   LIN {X 0.148, Y -17.815, Z 116.450} C_DIS
   LIN {X 0.105, Y -17.697, Z 116.450} C_DIS
   LIN {X 0.144, Y -15.870, Z 116.450} C_DIS
   LIN {X 0.185, Y -15.606, Z 116.450} C_DIS
   LIN {X 0.334, Y -15.400, Z 116.450} C_DIS
   LIN {X 1.468, Y -13.305, Z 116.450} C_DIS
   LIN {X 2.152, Y -12.926, Z 116.450} C_DIS
   LIN {X 3.732, Y -11.958, Z 116.450} C_DIS
   LIN {X 5.275, Y -11.875, Z 116.450} C_DIS
   LIN {X 5.904, Y -11.838, Z 116.450} C_DIS
   LIN {X 6.625, Y -12.128, Z 116.450} C_DIS
   LIN {X 7.876, Y -12.635, Z 116.450} C_DIS
   LIN {X 8.873, Y -13.791, Z 116.450} C_DIS
   LIN {X 9.540, Y -14.557, Z 116.450} C_DIS
   LIN {X 9.767, Y -15.717, Z 116.450}
   LaserEnd_Ext()
   LIN {X -10.909, Y 41.483, Z 116.450}
   LaserStart_Ext()
   LIN {X -11.006, Y 41.733, Z 116.450} C_DIS
   LIN {X -11.451, Y 43.299, Z 116.450} C_DIS
   LIN {X -10.985, Y 45.327, Z 116.450} C_DIS
   LIN {X -10.916, Y 45.490, Z 116.450} C_DIS
   LIN {X -10.671, Y 45.761, Z 116.450} C_DIS
   LIN {X -9.977, Y 46.585, Z 116.450} C_DIS
   LIN {X -9.388, Y 46.930, Z 116.450} C_DIS
   LIN {X -8.600, Y 47.307, Z 116.450} C_DIS
   LIN {X -8.343, Y 47.326, Z 116.450} C_DIS
   LIN {X -6.766, Y 47.399, Z 116.450} C_DIS
   LIN {X -6.451, Y 47.269, Z 116.450} C_DIS
   LIN {X -5.150, Y 46.712, Z 116.450} C_DIS
   LIN {X -4.172, Y 45.690, Z 116.450} C_DIS
   LIN {X -4.100, Y 45.595, Z 116.450} C_DIS
   LIN {X -3.202, Y 44.213, Z 116.450} C_DIS
   LIN {X -2.206, Y 42.575, Z 116.450} C_DIS
   LIN {X -1.280, Y 41.069, Z 116.450} C_DIS
   LIN {X 0.088, Y 38.632, Z 116.450} C_DIS
   LIN {X 0.776, Y 37.421, Z 116.450} C_DIS
   LIN {X 1.017, Y 36.980, Z 116.450} C_DIS
   LIN {X 3.124, Y 32.754, Z 116.450} C_DIS
   LIN {X 4.597, Y 29.710, Z 116.450} C_DIS
   LIN {X 5.895, Y 26.489, Z 116.450} C_DIS
   LIN {X 7.344, Y 22.915, Z 116.450} C_DIS
   LIN {X 8.835, Y 18.359, Z 116.450} C_DIS
   LIN {X 10.168, Y 14.012, Z 116.450} C_DIS
   LIN {X 11.828, Y 6.827, Z 116.450} C_DIS
   LIN {X 12.484, Y 3.575, Z 116.450} C_DIS
   LIN {X 13.461, Y -3.473, Z 116.450} C_DIS
   LIN {X 13.499, Y -3.785, Z 116.450} C_DIS
   LIN {X 13.808, Y -7.587, Z 116.450} C_DIS
   LIN {X 13.839, Y -7.818, Z 116.450} C_DIS
   LIN {X 13.902, Y -8.784, Z 116.450} C_DIS
   LIN {X 13.967, Y -10.194, Z 116.450} C_DIS
   LIN {X 14.021, Y -11.696, Z 116.450} C_DIS
   LIN {X 14.069, Y -13.595, Z 116.450} C_DIS
   LIN {X 14.061, Y -15.779, Z 116.450} C_DIS
   LIN {X 14.062, Y -16.860, Z 116.450} C_DIS
   LIN {X 13.686, Y -18.412, Z 116.450} C_DIS
   LIN {X 13.131, Y -20.708, Z 116.450} C_DIS
   LIN {X 12.132, Y -22.067, Z 116.450} C_DIS
   LIN {X 11.479, Y -23.029, Z 116.450} C_DIS
   LIN {X 10.917, Y -23.560, Z 116.450} C_DIS
   LIN {X 9.337, Y -24.637, Z 116.450} C_DIS
   LIN {X 8.125, Y -25.174, Z 116.450} C_DIS
   LIN {X 5.580, Y -25.760, Z 116.450} C_DIS
   LIN {X 4.678, Y -25.759, Z 116.450} C_DIS
   LIN {X 2.942, Y -25.575, Z 116.450} C_DIS
   LIN {X 2.640, Y -25.450, Z 116.450} C_DIS
   LIN {X -0.209, Y -24.162, Z 116.450} C_DIS
   LIN {X -0.493, Y -23.865, Z 116.450} C_DIS
   LIN {X -2.856, Y -21.202, Z 116.450} C_DIS
   LIN {X -3.165, Y -20.226, Z 116.450} C_DIS
   LIN {X -3.943, Y -17.598, Z 116.450} C_DIS
   LIN {X -3.816, Y -16.292, Z 116.450} C_DIS
   LIN {X -3.648, Y -14.441, Z 116.450} C_DIS
   LIN {X -2.859, Y -11.235, Z 116.450} C_DIS
   LIN {X -2.701, Y -10.616, Z 116.450} C_DIS
   LIN {X -2.627, Y -10.239, Z 116.450} C_DIS
   LIN {X -2.158, Y -7.884, Z 116.450} C_DIS
   LIN {X -1.604, Y -4.053, Z 116.450} C_DIS
   LIN {X -1.466, Y -3.109, Z 116.450} C_DIS
   LIN {X -1.367, Y -1.347, Z 116.450} C_DIS
   LIN {X -1.059, Y 3.657, Z 116.450} C_DIS
   LIN {X -1.134, Y 7.378, Z 116.450} C_DIS
   LIN {X -1.528, Y 13.286, Z 116.450} C_DIS
   LIN {X -2.342, Y 18.188, Z 116.450} C_DIS
   LIN {X -3.212, Y 22.624, Z 116.450} C_DIS
   LIN {X -4.479, Y 26.756, Z 116.450} C_DIS
   LIN {X -5.529, Y 30.144, Z 116.450} C_DIS
   LIN {X -5.798, Y 30.771, Z 116.450} C_DIS
   LIN {X -6.098, Y 31.534, Z 116.450} C_DIS
   LIN {X -7.395, Y 34.580, Z 116.450} C_DIS
   LIN {X -8.008, Y 35.958, Z 116.450} C_DIS
   LIN {X -8.997, Y 37.945, Z 116.450} C_DIS
   LIN {X -9.450, Y 38.841, Z 116.450} C_DIS
   LIN {X -10.064, Y 39.969, Z 116.450} C_DIS
   LIN {X -10.750, Y 41.198, Z 116.450} C_DIS
   LIN {X -10.909, Y 41.483, Z 116.450}
   LaserEnd_Ext()
   LIN {X 12.602, Y -5.091, Z 116.450}
   LaserStart_Ext()
   LIN {X 12.602, Y -18.640, Z 116.450}
   LaserEnd_Ext()
   LIN {X 11.602, Y -21.099, Z 116.450}
   LaserStart_Ext()
   LIN {X 11.602, Y 2.657, Z 116.450}
   LaserEnd_Ext()
   LIN {X 10.602, Y 7.690, Z 116.450}
   LaserStart_Ext()
   LIN {X 10.602, Y -14.776, Z 116.450}
   LaserEnd_Ext()
   LIN {X 10.602, Y -18.691, Z 116.450}
   LaserStart_Ext()
   LIN {X 10.602, Y -22.482, Z 116.450}
   LaserEnd_Ext()
   LIN {X 9.602, Y -23.246, Z 116.450}
   LaserStart_Ext()
   LIN {X 9.602, Y -20.491, Z 116.450}
   LaserEnd_Ext()
   LIN {X 9.602, Y -13.105, Z 116.450}
   LaserStart_Ext()
   LIN {X 9.602, Y 12.019, Z 116.450}
   LaserEnd_Ext()
   LIN {X 8.602, Y 15.708, Z 116.450}
   LaserStart_Ext()
   LIN {X 8.602, Y -11.949, Z 116.450}
   LaserEnd_Ext()
   LIN {X 8.602, Y -21.573, Z 116.450}
   LaserStart_Ext()
   LIN {X 8.602, Y -23.869, Z 116.450}
   LaserEnd_Ext()
   LIN {X 7.602, Y -24.269, Z 116.450}
   LaserStart_Ext()
   LIN {X 7.602, Y -22.068, Z 116.450}
   LaserEnd_Ext()
   LIN {X 7.602, Y -11.445, Z 116.450}
   LaserStart_Ext()
   LIN {X 7.602, Y 18.912, Z 116.450}
   LaserEnd_Ext()
   LIN {X 6.602, Y 21.967, Z 116.450}
   LaserStart_Ext()
   LIN {X 6.602, Y -11.041, Z 116.450}
   LaserEnd_Ext()
   LIN {X 6.602, Y -22.559, Z 116.450}
   LaserStart_Ext()
   LIN {X 6.602, Y -24.499, Z 116.450}
   LaserEnd_Ext()
   LIN {X 5.602, Y -24.728, Z 116.450}
   LaserStart_Ext()
   LIN {X 5.602, Y -22.670, Z 116.450}
   LaserEnd_Ext()
   LIN {X 5.602, Y -10.854, Z 116.450}
   LaserStart_Ext()
   LIN {X 5.602, Y 24.551, Z 116.450}
   LaserEnd_Ext()
   LIN {X 4.602, Y 27.023, Z 116.450}
   LaserStart_Ext()
   LIN {X 4.602, Y -10.910, Z 116.450}
   LaserEnd_Ext()
   LIN {X 4.602, Y -22.710, Z 116.450}
   LaserStart_Ext()
   LIN {X 4.602, Y -24.745, Z 116.450}
   LaserEnd_Ext()
   LIN {X 3.602, Y -24.639, Z 116.450}
   LaserStart_Ext()
   LIN {X 3.602, Y -22.581, Z 116.450}
   LaserEnd_Ext()
   LIN {X 3.602, Y -10.967, Z 116.450}
   LaserStart_Ext()
   LIN {X 3.602, Y 29.471, Z 116.450}
   LaserEnd_Ext()
   LIN {X 2.602, Y 31.537, Z 116.450}
   LaserStart_Ext()
   LIN {X 2.602, Y -11.477, Z 116.450}
   LaserEnd_Ext()
   LIN {X 2.602, Y -22.181, Z 116.450}
   LaserStart_Ext()
   LIN {X 2.602, Y -24.335, Z 116.450}
   LaserEnd_Ext()
   LIN {X 1.602, Y -23.883, Z 116.450}
   LaserStart_Ext()
   LIN {X 1.602, Y -21.731, Z 116.450}
   LaserEnd_Ext()
   LIN {X 1.602, Y -12.088, Z 116.450}
   LaserStart_Ext()
   LIN {X 1.602, Y 33.566, Z 116.450}
   LaserEnd_Ext()
   LIN {X 0.602, Y 35.571, Z 116.450}
   LaserStart_Ext()
   LIN {X 0.602, Y -12.808, Z 116.450}
   LaserEnd_Ext()
   LIN {X 0.602, Y -20.717, Z 116.450}
   LaserStart_Ext()
   LIN {X 0.602, Y -23.432, Z 116.450}
   LaserEnd_Ext()
   LIN {X -0.398, Y -22.465, Z 116.450}
   LaserStart_Ext()
   LIN {X -0.398, Y -19.184, Z 116.450}
   LaserEnd_Ext()
   LIN {X -0.398, Y -14.651, Z 116.450}
   LaserStart_Ext()
   LIN {X -0.398, Y -1.923, Z 116.450}
   LaserEnd_Ext()
   LIN {X -0.398, Y 11.377, Z 116.450}
   LaserStart_Ext()
   LIN {X -0.398, Y 37.462, Z 116.450}
   LaserEnd_Ext()
   LIN {X -1.398, Y 39.236, Z 116.450}
   LaserStart_Ext()
   LIN {X -1.398, Y 18.572, Z 116.450}
   LaserEnd_Ext()
   LIN {X -1.398, Y -9.189, Z 116.450}
   LaserStart_Ext()
   LIN {X -1.398, Y -21.338, Z 116.450}
   LaserEnd_Ext()
   LIN {X -2.398, Y -19.295, Z 116.450}
   LaserStart_Ext()
   LIN {X -2.398, Y -13.547, Z 116.450}
   LaserEnd_Ext()
   LIN {X -2.398, Y 23.380, Z 116.450}
   LaserStart_Ext()
   LIN {X -2.398, Y 40.979, Z 116.450}
   LaserEnd_Ext()
   LIN {X -3.398, Y 42.611, Z 116.450}
   LaserStart_Ext()
   LIN {X -3.398, Y 26.642, Z 116.450}
   LaserEnd_Ext()
   LIN {X -4.398, Y 29.872, Z 116.450}
   LaserStart_Ext()
   LIN {X -4.398, Y 44.218, Z 116.450}
   LaserEnd_Ext()
   LIN {X -5.398, Y 45.524, Z 116.450}
   LaserStart_Ext()
   LIN {X -5.398, Y 32.443, Z 116.450}
   LaserEnd_Ext()
   LIN {X -6.398, Y 34.792, Z 116.450}
   LaserStart_Ext()
   LIN {X -6.398, Y 46.158, Z 116.450}
   LaserEnd_Ext()
   LIN {X -7.398, Y 46.368, Z 116.450}
   LaserStart_Ext()
   LIN {X -7.398, Y 36.977, Z 116.450}
   LaserEnd_Ext()
   LIN {X -8.398, Y 38.977, Z 116.450}
   LaserStart_Ext()
   LIN {X -8.398, Y 46.295, Z 116.450}
   LaserEnd_Ext()
   LIN {X -9.398, Y 45.720, Z 116.450}
   LaserStart_Ext()
   LIN {X -9.398, Y 40.828, Z 116.450}
   LaserEnd_Ext()
   LIN {X -10.398, Y 43.252, Z 116.450}
   LaserStart_Ext()
   LIN {X -10.398, Y 43.501, Z 116.450}
   LaserEnd_Ext()
   LIN {X 2.352, Y -12.792, Z 117.300}
   LaserStart_Ext()
   LIN {X 3.808, Y -11.899, Z 117.300} C_DIS
   LIN {X 4.082, Y -11.884, Z 117.300} C_DIS
   LIN {X 5.981, Y -11.774, Z 117.300} C_DIS
   LIN {X 7.781, Y -12.497, Z 117.300} C_DIS
   LIN {X 7.954, Y -12.566, Z 117.300} C_DIS
   LIN {X 8.122, Y -12.758, Z 117.300} C_DIS
   LIN {X 9.624, Y -14.482, Z 117.300} C_DIS
   LIN {X 10.019, Y -16.502, Z 117.300} C_DIS
   LIN {X 10.117, Y -17.066, Z 117.300} C_DIS
   LIN {X 10.008, Y -17.325, Z 117.300} C_DIS
   LIN {X 9.461, Y -19.163, Z 117.300} C_DIS
   LIN {X 9.174, Y -19.483, Z 117.300} C_DIS
   LIN {X 8.261, Y -20.603, Z 117.300} C_DIS
   LIN {X 7.039, Y -21.215, Z 117.300} C_DIS
   LIN {X 6.305, Y -21.578, Z 117.300} C_DIS
   LIN {X 5.059, Y -21.630, Z 117.300} C_DIS
   LIN {X 4.256, Y -21.666, Z 117.300} C_DIS
   LIN {X 3.735, Y -21.461, Z 117.300} C_DIS
   LIN {X 2.335, Y -20.902, Z 117.300} C_DIS
   LIN {X 1.034, Y -19.575, Z 117.300} C_DIS
   LIN {X 0.886, Y -19.430, Z 117.300} C_DIS
   LIN {X 0.843, Y -19.336, Z 117.300} C_DIS
   LIN {X 0.209, Y -17.706, Z 117.300} C_DIS
   LIN {X 0.242, Y -16.089, Z 117.300} C_DIS
   LIN {X 0.232, Y -15.677, Z 117.300} C_DIS
   LIN {X 1.388, Y -13.470, Z 117.300} C_DIS
   LIN {X 1.506, Y -13.295, Z 117.300} C_DIS
   LIN {X 2.352, Y -12.792, Z 117.300}
   LaserEnd_Ext()
   LIN {X -10.228, Y 46.455, Z 117.300}
   LaserStart_Ext()
   LIN {X -8.835, Y 47.270, Z 117.300} C_DIS
   LIN {X -8.739, Y 47.316, Z 117.300} C_DIS
   LIN {X -7.015, Y 47.441, Z 117.300} C_DIS
   LIN {X -6.906, Y 47.446, Z 117.300} C_DIS
   LIN {X -5.837, Y 47.004, Z 117.300} C_DIS
   LIN {X -5.218, Y 46.751, Z 117.300} C_DIS
   LIN {X -4.194, Y 45.692, Z 117.300} C_DIS
   LIN {X -3.623, Y 44.809, Z 117.300} C_DIS
   LIN {X -3.110, Y 44.019, Z 117.300} C_DIS
   LIN {X -1.466, Y 41.317, Z 117.300} C_DIS
   LIN {X -1.246, Y 40.962, Z 117.300} C_DIS
   LIN {X -1.128, Y 40.764, Z 117.300} C_DIS
   LIN {X 0.502, Y 37.895, Z 117.300} C_DIS
   LIN {X 1.213, Y 36.595, Z 117.300} C_DIS
   LIN {X 2.850, Y 33.312, Z 117.300} C_DIS
   LIN {X 4.633, Y 29.628, Z 117.300} C_DIS
   LIN {X 5.665, Y 27.069, Z 117.300} C_DIS
   LIN {X 7.447, Y 22.670, Z 117.300} C_DIS
   LIN {X 8.661, Y 18.962, Z 117.300} C_DIS
   LIN {X 10.345, Y 13.469, Z 117.300} C_DIS
   LIN {X 11.735, Y 7.454, Z 117.300} C_DIS
   LIN {X 12.611, Y 3.117, Z 117.300} C_DIS
   LIN {X 13.446, Y -2.907, Z 117.300} C_DIS
   LIN {X 13.600, Y -4.184, Z 117.300} C_DIS
   LIN {X 13.868, Y -7.474, Z 117.300} C_DIS
   LIN {X 13.906, Y -7.768, Z 117.300} C_DIS
   LIN {X 13.987, Y -8.999, Z 117.300} C_DIS
   LIN {X 14.014, Y -9.585, Z 117.300} C_DIS
   LIN {X 14.134, Y -12.868, Z 117.300} C_DIS
   LIN {X 14.150, Y -13.509, Z 117.300} C_DIS
   LIN {X 14.147, Y -14.246, Z 117.300} C_DIS
   LIN {X 14.152, Y -16.774, Z 117.300} C_DIS
   LIN {X 13.271, Y -20.403, Z 117.300} C_DIS
   LIN {X 13.205, Y -20.676, Z 117.300} C_DIS
   LIN {X 13.086, Y -20.838, Z 117.300} C_DIS
   LIN {X 11.830, Y -22.691, Z 117.300} C_DIS
   LIN {X 10.750, Y -23.712, Z 117.300} C_DIS
   LIN {X 9.871, Y -24.310, Z 117.300} C_DIS
   LIN {X 7.645, Y -25.298, Z 117.300} C_DIS
   LIN {X 6.126, Y -25.647, Z 117.300} C_DIS
   LIN {X 4.190, Y -25.646, Z 117.300} C_DIS
   LIN {X 3.126, Y -25.533, Z 117.300} C_DIS
   LIN {X 1.700, Y -24.941, Z 117.300} C_DIS
   LIN {X -0.040, Y -24.154, Z 117.300} C_DIS
   LIN {X -1.305, Y -22.829, Z 117.300} C_DIS
   LIN {X -2.695, Y -21.263, Z 117.300} C_DIS
   LIN {X -3.641, Y -18.277, Z 117.300} C_DIS
   LIN {X -3.853, Y -17.560, Z 117.300} C_DIS
   LIN {X -3.818, Y -17.203, Z 117.300} C_DIS
   LIN {X -3.565, Y -14.402, Z 117.300} C_DIS
   LIN {X -2.820, Y -11.378, Z 117.300} C_DIS
   LIN {X -2.522, Y -10.037, Z 117.300} C_DIS
   LIN {X -2.151, Y -8.171, Z 117.300} C_DIS
   LIN {X -1.440, Y -3.250, Z 117.300} C_DIS
   LIN {X -1.418, Y -3.006, Z 117.300} C_DIS
   LIN {X -1.034, Y 3.218, Z 117.300} C_DIS
   LIN {X -1.127, Y 7.848, Z 117.300} C_DIS
   LIN {X -1.461, Y 12.849, Z 117.300} C_DIS
   LIN {X -2.442, Y 18.758, Z 117.300} C_DIS
   LIN {X -3.160, Y 22.418, Z 117.300} C_DIS
   LIN {X -4.659, Y 27.305, Z 117.300} C_DIS
   LIN {X -5.505, Y 30.034, Z 117.300} C_DIS
   LIN {X -5.809, Y 30.745, Z 117.300} C_DIS
   LIN {X -5.975, Y 31.166, Z 117.300} C_DIS
   LIN {X -7.620, Y 35.030, Z 117.300} C_DIS
   LIN {X -7.914, Y 35.691, Z 117.300} C_DIS
   LIN {X -9.253, Y 38.384, Z 117.300} C_DIS
   LIN {X -9.442, Y 38.756, Z 117.300} C_DIS
   LIN {X -9.697, Y 39.225, Z 117.300} C_DIS
   LIN {X -10.133, Y 40.006, Z 117.300} C_DIS
   LIN {X -10.961, Y 41.508, Z 117.300} C_DIS
   LIN {X -11.151, Y 42.020, Z 117.300} C_DIS
   LIN {X -11.490, Y 43.166, Z 117.300} C_DIS
   LIN {X -11.440, Y 43.879, Z 117.300} C_DIS
   LIN {X -11.089, Y 45.273, Z 117.300} C_DIS
   LIN {X -10.777, Y 45.775, Z 117.300} C_DIS
   LIN {X -10.454, Y 46.186, Z 117.300} C_DIS
   LIN {X -10.228, Y 46.455, Z 117.300}
   LaserEnd_Ext()
   LIN {X -9.705, Y 45.522, Z 117.300}
   LaserStart_Ext()
   LIN {X -5.421, Y 45.522, Z 117.300}
   LaserEnd_Ext()
   LIN {X -4.628, Y 44.522, Z 117.300}
   LaserStart_Ext()
   LIN {X -10.247, Y 44.522, Z 117.300}
   LaserEnd_Ext()
   LIN {X -10.463, Y 43.522, Z 117.300}
   LaserStart_Ext()
   LIN {X -3.979, Y 43.522, Z 117.300}
   LaserEnd_Ext()
   LIN {X -3.369, Y 42.522, Z 117.300}
   LaserStart_Ext()
   LIN {X -10.257, Y 42.522, Z 117.300}
   LaserEnd_Ext()
   LIN {X -9.827, Y 41.522, Z 117.300}
   LaserStart_Ext()
   LIN {X -2.761, Y 41.522, Z 117.300}
   LaserEnd_Ext()
   LIN {X -2.150, Y 40.522, Z 117.300}
   LaserStart_Ext()
   LIN {X -9.275, Y 40.522, Z 117.300}
   LaserEnd_Ext()
   LIN {X -8.720, Y 39.522, Z 117.300}
   LaserStart_Ext()
   LIN {X -1.573, Y 39.522, Z 117.300}
   LaserEnd_Ext()
   LIN {X -1.004, Y 38.522, Z 117.300}
   LaserStart_Ext()
   LIN {X -8.205, Y 38.522, Z 117.300}
   LaserEnd_Ext()
   LIN {X -7.708, Y 37.522, Z 117.300}
   LaserStart_Ext()
   LIN {X -0.436, Y 37.522, Z 117.300}
   LaserEnd_Ext()
   LIN {X 0.114, Y 36.522, Z 117.300}
   LaserStart_Ext()
   LIN {X -7.210, Y 36.522, Z 117.300}
   LaserEnd_Ext()
   LIN {X -6.744, Y 35.522, Z 117.300}
   LaserStart_Ext()
   LIN {X 0.631, Y 35.522, Z 117.300}
   LaserEnd_Ext()
   LIN {X 1.130, Y 34.522, Z 117.300}
   LaserStart_Ext()
   LIN {X -6.317, Y 34.522, Z 117.300}
   LaserEnd_Ext()
   LIN {X -5.891, Y 33.522, Z 117.300}
   LaserStart_Ext()
   LIN {X 1.628, Y 33.522, Z 117.300}
   LaserEnd_Ext()
   LIN {X 2.122, Y 32.522, Z 117.300}
   LaserStart_Ext()
   LIN {X -5.465, Y 32.522, Z 117.300}
   LaserEnd_Ext()
   LIN {X -5.040, Y 31.522, Z 117.300}
   LaserStart_Ext()
   LIN {X 2.606, Y 31.522, Z 117.300}
   LaserEnd_Ext()
   LIN {X 3.090, Y 30.522, Z 117.300}
   LaserStart_Ext()
   LIN {X -4.626, Y 30.522, Z 117.300}
   LaserEnd_Ext()
   LIN {X -4.299, Y 29.522, Z 117.300}
   LaserStart_Ext()
   LIN {X 3.574, Y 29.522, Z 117.300}
   LaserEnd_Ext()
   LIN {X 4.001, Y 28.522, Z 117.300}
   LaserStart_Ext()
   LIN {X -3.989, Y 28.522, Z 117.300}
   LaserEnd_Ext()
   LIN {X -3.679, Y 27.522, Z 117.300}
   LaserStart_Ext()
   LIN {X 4.404, Y 27.522, Z 117.300}
   LaserEnd_Ext()
   LIN {X 4.808, Y 26.522, Z 117.300}
   LaserStart_Ext()
   LIN {X -3.373, Y 26.522, Z 117.300}
   LaserEnd_Ext()
   LIN {X -3.066, Y 25.522, Z 117.300}
   LaserStart_Ext()
   LIN {X 5.213, Y 25.522, Z 117.300}
   LaserEnd_Ext()
   LIN {X 5.618, Y 24.522, Z 117.300}
   LaserStart_Ext()
   LIN {X -2.760, Y 24.522, Z 117.300}
   LaserEnd_Ext()
   LIN {X -2.453, Y 23.522, Z 117.300}
   LaserStart_Ext()
   LIN {X 6.023, Y 23.522, Z 117.300}
   LaserEnd_Ext()
   LIN {X 6.429, Y 22.522, Z 117.300}
   LaserStart_Ext()
   LIN {X -2.162, Y 22.522, Z 117.300}
   LaserEnd_Ext()
   LIN {X -1.966, Y 21.522, Z 117.300}
   LaserStart_Ext()
   LIN {X 6.771, Y 21.522, Z 117.300}
   LaserEnd_Ext()
   LIN {X 7.098, Y 20.522, Z 117.300}
   LaserStart_Ext()
   LIN {X -1.769, Y 20.522, Z 117.300}
   LaserEnd_Ext()
   LIN {X -1.573, Y 19.522, Z 117.300}
   LaserStart_Ext()
   LIN {X 7.426, Y 19.522, Z 117.300}
   LaserEnd_Ext()
   LIN {X 7.750, Y 18.522, Z 117.300}
   LaserStart_Ext()
   LIN {X -1.389, Y 18.522, Z 117.300}
   LaserEnd_Ext()
   LIN {X -1.223, Y 17.522, Z 117.300}
   LaserStart_Ext()
   LIN {X 8.057, Y 17.522, Z 117.300}
   LaserEnd_Ext()
   LIN {X 8.363, Y 16.522, Z 117.300}
   LaserStart_Ext()
   LIN {X -1.057, Y 16.522, Z 117.300}
   LaserEnd_Ext()
   LIN {X -0.891, Y 15.522, Z 117.300}
   LaserStart_Ext()
   LIN {X 8.670, Y 15.522, Z 117.300}
   LaserEnd_Ext()
   LIN {X 8.977, Y 14.522, Z 117.300}
   LaserStart_Ext()
   LIN {X -0.725, Y 14.522, Z 117.300}
   LaserEnd_Ext()
   LIN {X -0.559, Y 13.522, Z 117.300}
   LaserStart_Ext()
   LIN {X 9.283, Y 13.522, Z 117.300}
   LaserEnd_Ext()
   LIN {X 9.538, Y 12.522, Z 117.300}
   LaserStart_Ext()
   LIN {X -0.437, Y 12.522, Z 117.300}
   LaserEnd_Ext()
   LIN {X -0.370, Y 11.522, Z 117.300}
   LaserStart_Ext()
   LIN {X 9.769, Y 11.522, Z 117.300}
   LaserEnd_Ext()
   LIN {X 10.000, Y 10.522, Z 117.300}
   LaserStart_Ext()
   LIN {X -0.303, Y 10.522, Z 117.300}
   LaserEnd_Ext()
   LIN {X -0.237, Y 9.522, Z 117.300}
   LaserStart_Ext()
   LIN {X 10.231, Y 9.522, Z 117.300}
   LaserEnd_Ext()
   LIN {X 10.462, Y 8.522, Z 117.300}
   LaserStart_Ext()
   LIN {X -0.170, Y 8.522, Z 117.300}
   LaserEnd_Ext()
   LIN {X -0.120, Y 7.522, Z 117.300}
   LaserStart_Ext()
   LIN {X 10.693, Y 7.522, Z 117.300}
   LaserEnd_Ext()
   LIN {X 10.903, Y 6.522, Z 117.300}
   LaserStart_Ext()
   LIN {X -0.100, Y 6.522, Z 117.300}
   LaserEnd_Ext()
   LIN {X -0.080, Y 5.522, Z 117.300}
   LaserStart_Ext()
   LIN {X 11.105, Y 5.522, Z 117.300}
   LaserEnd_Ext()
   LIN {X 11.307, Y 4.522, Z 117.300}
   LaserStart_Ext()
   LIN {X -0.060, Y 4.522, Z 117.300}
   LaserEnd_Ext()
   LIN {X -0.040, Y 3.522, Z 117.300}
   LaserStart_Ext()
   LIN {X 11.509, Y 3.522, Z 117.300}
   LaserEnd_Ext()
   LIN {X 11.684, Y 2.522, Z 117.300}
   LaserStart_Ext()
   LIN {X -0.075, Y 2.522, Z 117.300}
   LaserEnd_Ext()
   LIN {X -0.137, Y 1.522, Z 117.300}
   LaserStart_Ext()
   LIN {X 11.822, Y 1.522, Z 117.300}
   LaserEnd_Ext()
   LIN {X 11.961, Y 0.522, Z 117.300}
   LaserStart_Ext()
   LIN {X -0.199, Y 0.522, Z 117.300}
   LaserEnd_Ext()
   LIN {X -0.260, Y -0.478, Z 117.300}
   LaserStart_Ext()
   LIN {X 12.099, Y -0.478, Z 117.300}
   LaserEnd_Ext()
   LIN {X 12.238, Y -1.478, Z 117.300}
   LaserStart_Ext()
   LIN {X -0.322, Y -1.478, Z 117.300}
   LaserEnd_Ext()
   LIN {X -0.384, Y -2.478, Z 117.300}
   LaserStart_Ext()
   LIN {X 12.377, Y -2.478, Z 117.300}
   LaserEnd_Ext()
   LIN {X 12.507, Y -3.478, Z 117.300}
   LaserStart_Ext()
   LIN {X -0.462, Y -3.478, Z 117.300}
   LaserEnd_Ext()
   LIN {X -0.607, Y -4.478, Z 117.300}
   LaserStart_Ext()
   LIN {X 12.620, Y -4.478, Z 117.300}
   LaserEnd_Ext()
   LIN {X 12.702, Y -5.478, Z 117.300}
   LaserStart_Ext()
   LIN {X -0.751, Y -5.478, Z 117.300}
   LaserEnd_Ext()
   LIN {X -0.896, Y -6.478, Z 117.300}
   LaserStart_Ext()
   LIN {X 12.783, Y -6.478, Z 117.300}
   LaserEnd_Ext()
   LIN {X 12.865, Y -7.478, Z 117.300}
   LaserStart_Ext()
   LIN {X -1.040, Y -7.478, Z 117.300}
   LaserEnd_Ext()
   LIN {X -1.193, Y -8.478, Z 117.300}
   LaserStart_Ext()
   LIN {X 12.951, Y -8.478, Z 117.300}
   LaserEnd_Ext()
   LIN {X 13.008, Y -9.478, Z 117.300}
   LaserStart_Ext()
   LIN {X -1.392, Y -9.478, Z 117.300}
   LaserEnd_Ext()
   LIN {X -1.596, Y -10.478, Z 117.300}
   LaserStart_Ext()
   LIN {X 13.046, Y -10.478, Z 117.300}
   LaserEnd_Ext()
   LIN {X 13.082, Y -11.478, Z 117.300}
   LaserStart_Ext()
   LIN {X 7.928, Y -11.478, Z 117.300}
   LaserEnd_Ext()
   LIN {X 2.581, Y -11.478, Z 117.300}
   LaserStart_Ext()
   LIN {X -1.818, Y -11.478, Z 117.300}
   LaserEnd_Ext()
   LIN {X -2.061, Y -12.478, Z 117.300}
   LaserStart_Ext()
   LIN {X 0.932, Y -12.478, Z 117.300}
   LaserEnd_Ext()
   LIN {X 9.205, Y -12.478, Z 117.300}
   LaserStart_Ext()
   LIN {X 13.119, Y -12.478, Z 117.300}
   LaserEnd_Ext()
   LIN {X 13.149, Y -13.478, Z 117.300}
   LaserStart_Ext()
   LIN {X 10.076, Y -13.478, Z 117.300}
   LaserEnd_Ext()
   LIN {X 0.255, Y -13.478, Z 117.300}
   LaserStart_Ext()
   LIN {X -2.308, Y -13.478, Z 117.300}
   LaserEnd_Ext()
   LIN {X -2.554, Y -14.478, Z 117.300}
   LaserStart_Ext()
   LIN {X -0.269, Y -14.478, Z 117.300}
   LaserEnd_Ext()
   LIN {X 10.643, Y -14.478, Z 117.300}
   LaserStart_Ext()
   LIN {X 13.147, Y -14.478, Z 117.300}
   LaserEnd_Ext()
   LIN {X 13.149, Y -15.478, Z 117.300}
   LaserStart_Ext()
   LIN {X 10.838, Y -15.478, Z 117.300}
   LaserEnd_Ext()
   LIN {X -0.747, Y -15.478, Z 117.300}
   LaserStart_Ext()
   LIN {X -2.658, Y -15.478, Z 117.300}
   LaserEnd_Ext()
   LIN {X -2.749, Y -16.478, Z 117.300}
   LaserStart_Ext()
   LIN {X -0.766, Y -16.478, Z 117.300}
   LaserEnd_Ext()
   LIN {X 11.030, Y -16.478, Z 117.300}
   LaserStart_Ext()
   LIN {X 13.151, Y -16.478, Z 117.300}
   LaserEnd_Ext()
   LIN {X 12.952, Y -17.478, Z 117.300}
   LaserStart_Ext()
   LIN {X 11.029, Y -17.478, Z 117.300}
   LaserEnd_Ext()
   LIN {X -0.787, Y -17.478, Z 117.300}
   LaserStart_Ext()
   LIN {X -2.834, Y -17.478, Z 117.300}
   LaserEnd_Ext()
   LIN {X -2.528, Y -18.478, Z 117.300}
   LaserStart_Ext()
   LIN {X -0.564, Y -18.478, Z 117.300}
   LaserEnd_Ext()
   LIN {X 10.708, Y -18.478, Z 117.300}
   LaserStart_Ext()
   LIN {X 12.709, Y -18.478, Z 117.300}
   LaserEnd_Ext()
   LIN {X 12.466, Y -19.478, Z 117.300}
   LaserStart_Ext()
   LIN {X 10.408, Y -19.478, Z 117.300}
   LaserEnd_Ext()
   LIN {X -0.175, Y -19.478, Z 117.300}
   LaserStart_Ext()
   LIN {X -2.211, Y -19.478, Z 117.300}
   LaserEnd_Ext()
   LIN {X -1.894, Y -20.478, Z 117.300}
   LaserStart_Ext()
   LIN {X 0.519, Y -20.478, Z 117.300}
   LaserEnd_Ext()
   LIN {X 9.654, Y -20.478, Z 117.300}
   LaserStart_Ext()
   LIN {X 12.122, Y -20.478, Z 117.300}
   LaserEnd_Ext()
   LIN {X 11.444, Y -21.478, Z 117.300}
   LaserStart_Ext()
   LIN {X 8.743, Y -21.478, Z 117.300}
   LaserEnd_Ext()
   LIN {X 1.499, Y -21.478, Z 117.300}
   LaserStart_Ext()
   LIN {X -1.167, Y -21.478, Z 117.300}
   LaserEnd_Ext()
   LIN {X -0.257, Y -22.478, Z 117.300}
   LaserStart_Ext()
   LIN {X 3.590, Y -22.478, Z 117.300}
   LaserEnd_Ext()
   LIN {X 6.739, Y -22.478, Z 117.300}
   LaserStart_Ext()
   LIN {X 10.599, Y -22.478, Z 117.300}
   LaserEnd_Ext()
   LIN {X 9.280, Y -23.478, Z 117.300}
   LaserStart_Ext()
   LIN {X 0.893, Y -23.478, Z 117.300}
   LaserEnd_Ext()
   LIN {X 3.194, Y -24.478, Z 117.300}
   LaserStart_Ext()
   LIN {X 6.746, Y -24.478, Z 117.300}
   LaserEnd_Ext()
   LIN {X 0.313, Y -17.714, Z 118.150}
   LaserStart_Ext()
   LIN {X 0.334, Y -16.738, Z 118.150} C_DIS
   LIN {X 0.308, Y -15.682, Z 118.150} C_DIS
   LIN {X 1.008, Y -14.345, Z 118.150} C_DIS
   LIN {X 2.010, Y -12.865, Z 118.150} C_DIS
   LIN {X 3.097, Y -12.217, Z 118.150} C_DIS
   LIN {X 3.918, Y -11.830, Z 118.150} C_DIS
   LIN {X 5.248, Y -11.756, Z 118.150} C_DIS
   LIN {X 6.058, Y -11.709, Z 118.150} C_DIS
   LIN {X 6.630, Y -11.939, Z 118.150} C_DIS
   LIN {X 8.032, Y -12.495, Z 118.150} C_DIS
   LIN {X 9.401, Y -14.055, Z 118.150} C_DIS
   LIN {X 9.709, Y -14.408, Z 118.150} C_DIS
   LIN {X 9.789, Y -14.821, Z 118.150} C_DIS
   LIN {X 10.194, Y -17.137, Z 118.150} C_DIS
   LIN {X 9.743, Y -18.204, Z 118.150} C_DIS
   LIN {X 9.411, Y -19.321, Z 118.150} C_DIS
   LIN {X 8.712, Y -20.103, Z 118.150} C_DIS
   LIN {X 8.363, Y -20.531, Z 118.150} C_DIS
   LIN {X 7.118, Y -21.154, Z 118.150} C_DIS
   LIN {X 6.407, Y -21.512, Z 118.150} C_DIS
   LIN {X 5.965, Y -21.534, Z 118.150} C_DIS
   LIN {X 4.359, Y -21.605, Z 118.150} C_DIS
   LIN {X 2.590, Y -20.909, Z 118.150} C_DIS
   LIN {X 2.435, Y -20.847, Z 118.150} C_DIS
   LIN {X 2.291, Y -20.700, Z 118.150} C_DIS
   LIN {X 1.060, Y -19.489, Z 118.150} C_DIS
   LIN {X 0.696, Y -18.699, Z 118.150} C_DIS
   LIN {X 0.313, Y -17.714, Z 118.150}
   LaserEnd_Ext()
   LIN {X 5.434, Y 27.648, Z 118.150}
   LaserStart_Ext()
   LIN {X 7.551, Y 22.426, Z 118.150} C_DIS
   LIN {X 8.487, Y 19.565, Z 118.150} C_DIS
   LIN {X 10.523, Y 12.926, Z 118.150} C_DIS
   LIN {X 11.642, Y 8.081, Z 118.150} C_DIS
   LIN {X 12.737, Y 2.659, Z 118.150} C_DIS
   LIN {X 13.430, Y -2.341, Z 118.150} C_DIS
   LIN {X 13.701, Y -4.583, Z 118.150} C_DIS
   LIN {X 13.927, Y -7.360, Z 118.150} C_DIS
   LIN {X 13.974, Y -7.717, Z 118.150} C_DIS
   LIN {X 14.057, Y -8.977, Z 118.150} C_DIS
   LIN {X 14.084, Y -9.487, Z 118.150} C_DIS
   LIN {X 14.227, Y -13.327, Z 118.150} C_DIS
   LIN {X 14.236, Y -14.021, Z 118.150} C_DIS
   LIN {X 14.241, Y -16.688, Z 118.150} C_DIS
   LIN {X 13.561, Y -19.491, Z 118.150} C_DIS
   LIN {X 13.277, Y -20.645, Z 118.150} C_DIS
   LIN {X 12.211, Y -22.271, Z 118.150} C_DIS
   LIN {X 11.992, Y -22.543, Z 118.150} C_DIS
   LIN {X 11.243, Y -23.239, Z 118.150} C_DIS
   LIN {X 10.582, Y -23.864, Z 118.150} C_DIS
   LIN {X 10.405, Y -23.984, Z 118.150} C_DIS
   LIN {X 7.166, Y -25.421, Z 118.150} C_DIS
   LIN {X 6.673, Y -25.534, Z 118.150} C_DIS
   LIN {X 3.702, Y -25.533, Z 118.150} C_DIS
   LIN {X 3.311, Y -25.491, Z 118.150} C_DIS
   LIN {X 0.761, Y -24.432, Z 118.150} C_DIS
   LIN {X 0.129, Y -24.146, Z 118.150} C_DIS
   LIN {X -2.116, Y -21.794, Z 118.150} C_DIS
   LIN {X -2.534, Y -21.323, Z 118.150} C_DIS
   LIN {X -3.017, Y -19.799, Z 118.150} C_DIS
   LIN {X -3.747, Y -17.636, Z 118.150} C_DIS
   LIN {X -3.677, Y -16.521, Z 118.150} C_DIS
   LIN {X -3.482, Y -14.362, Z 118.150} C_DIS
   LIN {X -3.054, Y -12.626, Z 118.150} C_DIS
   LIN {X -2.279, Y -9.133, Z 118.150} C_DIS
   LIN {X -2.144, Y -8.459, Z 118.150} C_DIS
   LIN {X -1.863, Y -6.516, Z 118.150} C_DIS
   LIN {X -1.430, Y -3.566, Z 118.150} C_DIS
   LIN {X -1.344, Y -2.643, Z 118.150} C_DIS
   LIN {X -1.010, Y 2.780, Z 118.150} C_DIS
   LIN {X -1.121, Y 8.317, Z 118.150} C_DIS
   LIN {X -1.394, Y 12.412, Z 118.150} C_DIS
   LIN {X -2.543, Y 19.329, Z 118.150} C_DIS
   LIN {X -3.109, Y 22.211, Z 118.150} C_DIS
   LIN {X -4.839, Y 27.854, Z 118.150} C_DIS
   LIN {X -5.480, Y 29.924, Z 118.150} C_DIS
   LIN {X -5.821, Y 30.719, Z 118.150} C_DIS
   LIN {X -7.315, Y 34.235, Z 118.150} C_DIS
   LIN {X -7.814, Y 35.414, Z 118.150} C_DIS
   LIN {X -7.860, Y 35.509, Z 118.150} C_DIS
   LIN {X -9.384, Y 38.588, Z 118.150} C_DIS
   LIN {X -9.512, Y 38.827, Z 118.150} C_DIS
   LIN {X -10.087, Y 39.857, Z 118.150} C_DIS
   LIN {X -11.012, Y 41.533, Z 118.150} C_DIS
   LIN {X -11.438, Y 42.682, Z 118.150} C_DIS
   LIN {X -11.521, Y 42.964, Z 118.150} C_DIS
   LIN {X -11.416, Y 44.440, Z 118.150} C_DIS
   LIN {X -11.271, Y 45.016, Z 118.150} C_DIS
   LIN {X -10.554, Y 46.172, Z 118.150} C_DIS
   LIN {X -10.372, Y 46.405, Z 118.150} C_DIS
   LIN {X -9.427, Y 46.995, Z 118.150} C_DIS
   LIN {X -8.868, Y 47.325, Z 118.150} C_DIS
   LIN {X -7.586, Y 47.452, Z 118.150} C_DIS
   LIN {X -7.038, Y 47.493, Z 118.150} C_DIS
   LIN {X -5.790, Y 47.013, Z 118.150} C_DIS
   LIN {X -5.308, Y 46.815, Z 118.150} C_DIS
   LIN {X -4.290, Y 45.772, Z 118.150} C_DIS
   LIN {X -3.086, Y 43.932, Z 118.150} C_DIS
   LIN {X -3.017, Y 43.825, Z 118.150} C_DIS
   LIN {X -2.795, Y 43.460, Z 118.150} C_DIS
   LIN {X -1.560, Y 41.463, Z 118.150} C_DIS
   LIN {X -0.896, Y 40.347, Z 118.150} C_DIS
   LIN {X 0.228, Y 38.369, Z 118.150} C_DIS
   LIN {X 1.410, Y 36.211, Z 118.150} C_DIS
   LIN {X 2.576, Y 33.871, Z 118.150} C_DIS
   LIN {X 4.670, Y 29.545, Z 118.150} C_DIS
   LIN {X 5.434, Y 27.648, Z 118.150}
   LaserEnd_Ext()
   LIN {X -10.280, Y 44.717, Z 118.150}
   LaserStart_Ext()
   LIN {X -10.280, Y 42.436, Z 118.150}
   LaserEnd_Ext()
   LIN {X -9.280, Y 40.464, Z 118.150}
   LaserStart_Ext()
   LIN {X -9.280, Y 45.908, Z 118.150}
   LaserEnd_Ext()
   LIN {X -8.280, Y 46.378, Z 118.150}
   LaserStart_Ext()
   LIN {X -8.280, Y 38.611, Z 118.150}
   LaserEnd_Ext()
   LIN {X -7.280, Y 36.591, Z 118.150}
   LaserStart_Ext()
   LIN {X -7.280, Y 46.472, Z 118.150}
   LaserEnd_Ext()
   LIN {X -6.280, Y 46.130, Z 118.150}
   LaserStart_Ext()
   LIN {X -6.280, Y 34.356, Z 118.150}
   LaserEnd_Ext()
   LIN {X -5.280, Y 32.007, Z 118.150}
   LaserStart_Ext()
   LIN {X -5.280, Y 45.354, Z 118.150}
   LaserEnd_Ext()
   LIN {X -4.280, Y 43.935, Z 118.150}
   LaserStart_Ext()
   LIN {X -4.280, Y 29.428, Z 118.150}
   LaserEnd_Ext()
   LIN {X -3.280, Y 26.181, Z 118.150}
   LaserStart_Ext()
   LIN {X -3.280, Y 42.343, Z 118.150}
   LaserEnd_Ext()
   LIN {X -2.280, Y 40.717, Z 118.150}
   LaserStart_Ext()
   LIN {X -2.280, Y 22.919, Z 118.150}
   LaserEnd_Ext()
   LIN {X -2.280, Y -13.664, Z 118.150}
   LaserStart_Ext()
   LIN {X -2.280, Y -18.856, Z 118.150}
   LaserEnd_Ext()
   LIN {X -1.280, Y -21.222, Z 118.150}
   LaserStart_Ext()
   LIN {X -1.280, Y -9.238, Z 118.150}
   LaserEnd_Ext()
   LIN {X -1.280, Y 17.827, Z 118.150}
   LaserStart_Ext()
   LIN {X -1.280, Y 38.999, Z 118.150}
   LaserEnd_Ext()
   LIN {X -0.280, Y 37.215, Z 118.150}
   LaserStart_Ext()
   LIN {X -0.280, Y 10.732, Z 118.150}
   LaserEnd_Ext()
   LIN {X -0.280, Y -1.630, Z 118.150}
   LaserStart_Ext()
   LIN {X -0.280, Y -14.650, Z 118.150}
   LaserEnd_Ext()
   LIN {X -0.280, Y -18.948, Z 118.150}
   LaserStart_Ext()
   LIN {X -0.280, Y -22.269, Z 118.150}
   LaserEnd_Ext()
   LIN {X 0.720, Y -23.316, Z 118.150}
   LaserStart_Ext()
   LIN {X 0.720, Y -20.558, Z 118.150}
   LaserEnd_Ext()
   LIN {X 0.720, Y -12.987, Z 118.150}
   LaserStart_Ext()
   LIN {X 0.720, Y 35.353, Z 118.150}
   LaserEnd_Ext()
   LIN {X 1.720, Y 33.344, Z 118.150}
   LaserStart_Ext()
   LIN {X 1.720, Y -11.874, Z 118.150}
   LaserEnd_Ext()
   LIN {X 1.720, Y -21.546, Z 118.150}
   LaserStart_Ext()
   LIN {X 1.720, Y -23.747, Z 118.150}
   LaserEnd_Ext()
   LIN {X 2.720, Y -24.163, Z 118.150}
   LaserStart_Ext()
   LIN {X 2.720, Y -22.035, Z 118.150}
   LaserEnd_Ext()
   LIN {X 2.720, Y -11.290, Z 118.150}
   LaserStart_Ext()
   LIN {X 2.720, Y 31.278, Z 118.150}
   LaserEnd_Ext()
   LIN {X 3.720, Y 29.212, Z 118.150}
   LaserStart_Ext()
   LIN {X 3.720, Y -10.851, Z 118.150}
   LaserEnd_Ext()
   LIN {X 3.720, Y -22.428, Z 118.150}
   LaserStart_Ext()
   LIN {X 3.720, Y -24.529, Z 118.150}
   LaserEnd_Ext()
   LIN {X 4.720, Y -24.533, Z 118.150}
   LaserStart_Ext()
   LIN {X 4.720, Y -22.590, Z 118.150}
   LaserEnd_Ext()
   LIN {X 4.720, Y -10.784, Z 118.150}
   LaserStart_Ext()
   LIN {X 4.720, Y 26.748, Z 118.150}
   LaserEnd_Ext()
   LIN {X 5.720, Y 24.280, Z 118.150}
   LaserStart_Ext()
   LIN {X 5.720, Y -10.727, Z 118.150}
   LaserEnd_Ext()
   LIN {X 5.720, Y -22.546, Z 118.150}
   LaserStart_Ext()
   LIN {X 5.720, Y -24.534, Z 118.150}
   LaserEnd_Ext()
   LIN {X 6.720, Y -24.497, Z 118.150}
   LaserStart_Ext()
   LIN {X 6.720, Y -22.460, Z 118.150}
   LaserEnd_Ext()
   LIN {X 6.720, Y -10.897, Z 118.150}
   LaserStart_Ext()
   LIN {X 6.720, Y 21.749, Z 118.150}
   LaserEnd_Ext()
   LIN {X 7.720, Y 18.655, Z 118.150}
   LaserStart_Ext()
   LIN {X 7.720, Y -11.295, Z 118.150}
   LaserEnd_Ext()
   LIN {X 7.720, Y -21.971, Z 118.150}
   LaserStart_Ext()
   LIN {X 7.720, Y -24.081, Z 118.150}
   LaserEnd_Ext()
   LIN {X 8.720, Y -23.637, Z 118.150}
   LaserStart_Ext()
   LIN {X 8.720, Y -21.471, Z 118.150}
   LaserEnd_Ext()
   LIN {X 8.720, Y -11.770, Z 118.150}
   LaserStart_Ext()
   LIN {X 8.720, Y 15.394, Z 118.150}
   LaserEnd_Ext()
   LIN {X 9.720, Y 11.958, Z 118.150}
   LaserStart_Ext()
   LIN {X 9.720, Y -12.902, Z 118.150}
   LaserEnd_Ext()
   LIN {X 9.720, Y -20.476, Z 118.150}
   LaserStart_Ext()
   LIN {X 9.720, Y -23.194, Z 118.150}
   LaserEnd_Ext()
   LIN {X 10.720, Y -22.360, Z 118.150}
   LaserStart_Ext()
   LIN {X 10.720, Y -18.461, Z 118.150}
   LaserEnd_Ext()
   LIN {X 10.720, Y -14.370, Z 118.150}
   LaserStart_Ext()
   LIN {X 10.720, Y 7.594, Z 118.150}
   LaserEnd_Ext()
   LIN {X 11.720, Y 2.642, Z 118.150}
   LaserStart_Ext()
   LIN {X 11.720, Y -21.196, Z 118.150}
   LaserEnd_Ext()
   LIN {X 12.720, Y -18.714, Z 118.150}
   LaserStart_Ext()
   LIN {X 12.720, Y -4.863, Z 118.150}
   LaserEnd_Ext()
   LIN {X 4.462, Y -21.544, Z 119.000}
   LaserStart_Ext()
   LIN {X 3.989, Y -21.358, Z 119.000} C_DIS
   LIN {X 2.535, Y -20.791, Z 119.000} C_DIS
   LIN {X 1.714, Y -20.021, Z 119.000} C_DIS
   LIN {X 1.233, Y -19.548, Z 119.000} C_DIS
   LIN {X 0.550, Y -18.062, Z 119.000} C_DIS
   LIN {X 0.418, Y -17.723, Z 119.000} C_DIS
   LIN {X 0.425, Y -17.386, Z 119.000} C_DIS
   LIN {X 0.384, Y -15.688, Z 119.000} C_DIS
   LIN {X 0.629, Y -15.220, Z 119.000} C_DIS
   LIN {X 1.786, Y -13.510, Z 119.000} C_DIS
   LIN {X 2.286, Y -12.677, Z 119.000} C_DIS
   LIN {X 2.419, Y -12.519, Z 119.000} C_DIS
   LIN {X 2.710, Y -12.385, Z 119.000} C_DIS
   LIN {X 4.038, Y -11.759, Z 119.000} C_DIS
   LIN {X 5.465, Y -11.679, Z 119.000} C_DIS
   LIN {X 6.133, Y -11.644, Z 119.000} C_DIS
   LIN {X 6.997, Y -11.983, Z 119.000} C_DIS
   LIN {X 8.111, Y -12.425, Z 119.000} C_DIS
   LIN {X 8.919, Y -13.346, Z 119.000} C_DIS
   LIN {X 9.763, Y -14.283, Z 119.000} C_DIS
   LIN {X 9.901, Y -14.714, Z 119.000} C_DIS
   LIN {X 10.136, Y -16.440, Z 119.000} C_DIS
   LIN {X 10.270, Y -17.208, Z 119.000} C_DIS
   LIN {X 9.479, Y -19.083, Z 119.000} C_DIS
   LIN {X 9.361, Y -19.479, Z 119.000} C_DIS
   LIN {X 8.797, Y -20.110, Z 119.000} C_DIS
   LIN {X 8.443, Y -20.475, Z 119.000} C_DIS
   LIN {X 8.033, Y -20.678, Z 119.000} C_DIS
   LIN {X 6.509, Y -21.446, Z 119.000} C_DIS
   LIN {X 4.819, Y -21.529, Z 119.000} C_DIS
   LIN {X 4.462, Y -21.544, Z 119.000}
   LaserEnd_Ext()
   LIN {X -4.906, Y 46.398, Z 119.000}
   LaserStart_Ext()
   LIN {X -4.295, Y 45.777, Z 119.000} C_DIS
   LIN {X -3.832, Y 45.069, Z 119.000} C_DIS
   LIN {X -3.206, Y 44.101, Z 119.000} C_DIS
   LIN {X -2.641, Y 43.205, Z 119.000} C_DIS
   LIN {X -1.874, Y 41.964, Z 119.000} C_DIS
   LIN {X -0.663, Y 39.931, Z 119.000} C_DIS
   LIN {X -0.045, Y 38.843, Z 119.000} C_DIS
   LIN {X 1.606, Y 35.826, Z 119.000} C_DIS
   LIN {X 2.302, Y 34.429, Z 119.000} C_DIS
   LIN {X 4.706, Y 29.462, Z 119.000} C_DIS
   LIN {X 5.204, Y 28.228, Z 119.000} C_DIS
   LIN {X 7.654, Y 22.181, Z 119.000} C_DIS
   LIN {X 8.313, Y 20.167, Z 119.000} C_DIS
   LIN {X 10.701, Y 12.382, Z 119.000} C_DIS
   LIN {X 11.549, Y 8.709, Z 119.000} C_DIS
   LIN {X 12.863, Y 2.201, Z 119.000} C_DIS
   LIN {X 13.414, Y -1.775, Z 119.000} C_DIS
   LIN {X 13.802, Y -4.982, Z 119.000} C_DIS
   LIN {X 13.986, Y -7.246, Z 119.000} C_DIS
   LIN {X 14.041, Y -7.667, Z 119.000} C_DIS
   LIN {X 14.088, Y -8.372, Z 119.000} C_DIS
   LIN {X 14.211, Y -10.655, Z 119.000} C_DIS
   LIN {X 14.299, Y -13.047, Z 119.000} C_DIS
   LIN {X 14.327, Y -15.153, Z 119.000} C_DIS
   LIN {X 14.330, Y -16.602, Z 119.000} C_DIS
   LIN {X 13.960, Y -18.125, Z 119.000} C_DIS
   LIN {X 13.349, Y -20.613, Z 119.000} C_DIS
   LIN {X 12.662, Y -21.662, Z 119.000} C_DIS
   LIN {X 11.711, Y -22.840, Z 119.000} C_DIS
   LIN {X 10.690, Y -23.789, Z 119.000} C_DIS
   LIN {X 9.828, Y -24.218, Z 119.000} C_DIS
   LIN {X 7.053, Y -25.432, Z 119.000} C_DIS
   LIN {X 6.438, Y -25.459, Z 119.000} C_DIS
   LIN {X 3.513, Y -25.451, Z 119.000} C_DIS
   LIN {X 3.043, Y -25.280, Z 119.000} C_DIS
   LIN {X 0.314, Y -24.147, Z 119.000} C_DIS
   LIN {X -0.118, Y -23.734, Z 119.000} C_DIS
   LIN {X -2.372, Y -21.382, Z 119.000} C_DIS
   LIN {X -2.661, Y -20.657, Z 119.000} C_DIS
   LIN {X -3.632, Y -17.783, Z 119.000} C_DIS
   LIN {X -3.449, Y -14.880, Z 119.000} C_DIS
   LIN {X -3.399, Y -14.323, Z 119.000} C_DIS
   LIN {X -3.288, Y -13.875, Z 119.000} C_DIS
   LIN {X -2.822, Y -11.776, Z 119.000} C_DIS
   LIN {X -2.146, Y -8.772, Z 119.000} C_DIS
   LIN {X -2.086, Y -8.416, Z 119.000} C_DIS
   LIN {X -1.438, Y -4.006, Z 119.000} C_DIS
   LIN {X -1.256, Y -2.057, Z 119.000} C_DIS
   LIN {X -0.985, Y 2.342, Z 119.000} C_DIS
   LIN {X -1.115, Y 8.786, Z 119.000} C_DIS
   LIN {X -1.327, Y 11.974, Z 119.000} C_DIS
   LIN {X -2.644, Y 19.900, Z 119.000} C_DIS
   LIN {X -3.057, Y 22.004, Z 119.000} C_DIS
   LIN {X -5.018, Y 28.403, Z 119.000} C_DIS
   LIN {X -5.456, Y 29.814, Z 119.000} C_DIS
   LIN {X -5.713, Y 30.413, Z 119.000} C_DIS
   LIN {X -6.274, Y 31.785, Z 119.000} C_DIS
   LIN {X -7.649, Y 35.032, Z 119.000} C_DIS
   LIN {X -8.263, Y 36.312, Z 119.000} C_DIS
   LIN {X -9.204, Y 38.212, Z 119.000} C_DIS
   LIN {X -9.774, Y 39.281, Z 119.000} C_DIS
   LIN {X -10.785, Y 41.091, Z 119.000} C_DIS
   LIN {X -11.054, Y 41.562, Z 119.000} C_DIS
   LIN {X -11.390, Y 42.470, Z 119.000} C_DIS
   LIN {X -11.557, Y 42.919, Z 119.000} C_DIS
   LIN {X -11.510, Y 43.620, Z 119.000} C_DIS
   LIN {X -11.415, Y 44.832, Z 119.000} C_DIS
   LIN {X -11.197, Y 45.200, Z 119.000} C_DIS
   LIN {X -10.463, Y 46.393, Z 119.000} C_DIS
   LIN {X -9.953, Y 46.725, Z 119.000} C_DIS
   LIN {X -8.971, Y 47.342, Z 119.000} C_DIS
   LIN {X -8.203, Y 47.432, Z 119.000} C_DIS
   LIN {X -7.141, Y 47.538, Z 119.000} C_DIS
   LIN {X -6.354, Y 47.252, Z 119.000} C_DIS
   LIN {X -5.390, Y 46.881, Z 119.000} C_DIS
   LIN {X -4.906, Y 46.398, Z 119.000}
   LaserEnd_Ext()
   LIN {X 7.008, Y -24.360, Z 119.000}
   LaserStart_Ext()
   LIN {X 3.438, Y -24.360, Z 119.000}
   LaserEnd_Ext()
   LIN {X 1.027, Y -23.360, Z 119.000}
   LaserStart_Ext()
   LIN {X 9.293, Y -23.360, Z 119.000}
   LaserEnd_Ext()
   LIN {X 10.759, Y -22.360, Z 119.000}
   LaserStart_Ext()
   LIN {X 6.911, Y -22.360, Z 119.000}
   LaserEnd_Ext()
   LIN {X 3.804, Y -22.360, Z 119.000}
   LaserStart_Ext()
   LIN {X -0.049, Y -22.360, Z 119.000}
   LaserEnd_Ext()
   LIN {X -1.007, Y -21.360, Z 119.000}
   LaserStart_Ext()
   LIN {X 1.680, Y -21.360, Z 119.000}
   LaserEnd_Ext()
   LIN {X 8.906, Y -21.360, Z 119.000}
   LaserStart_Ext()
   LIN {X 11.620, Y -21.360, Z 119.000}
   LaserEnd_Ext()
   LIN {X 12.319, Y -20.360, Z 119.000}
   LaserStart_Ext()
   LIN {X 9.915, Y -20.360, Z 119.000}
   LaserEnd_Ext()
   LIN {X 0.632, Y -20.360, Z 119.000}
   LaserStart_Ext()
   LIN {X -1.703, Y -20.360, Z 119.000}
   LaserEnd_Ext()
   LIN {X -2.044, Y -19.360, Z 119.000}
   LaserStart_Ext()
   LIN {X 0.046, Y -19.360, Z 119.000}
   LaserEnd_Ext()
   LIN {X 10.447, Y -19.360, Z 119.000}
   LaserStart_Ext()
   LIN {X 12.627, Y -19.360, Z 119.000}
   LaserEnd_Ext()
   LIN {X 12.873, Y -18.360, Z 119.000}
   LaserStart_Ext()
   LIN {X 10.869, Y -18.360, Z 119.000}
   LaserEnd_Ext()
   LIN {X -0.407, Y -18.360, Z 119.000}
   LaserStart_Ext()
   LIN {X -2.382, Y -18.360, Z 119.000}
   LaserEnd_Ext()
   LIN {X -2.604, Y -17.360, Z 119.000}
   LaserStart_Ext()
   LIN {X -0.576, Y -17.360, Z 119.000}
   LaserEnd_Ext()
   LIN {X 11.257, Y -17.360, Z 119.000}
   LaserStart_Ext()
   LIN {X 13.117, Y -17.360, Z 119.000}
   LaserEnd_Ext()
   LIN {X 13.329, Y -16.360, Z 119.000}
   LaserStart_Ext()
   LIN {X 11.137, Y -16.360, Z 119.000}
   LaserEnd_Ext()
   LIN {X -0.600, Y -16.360, Z 119.000}
   LaserStart_Ext()
   LIN {X -2.540, Y -16.360, Z 119.000}
   LaserEnd_Ext()
   LIN {X -2.477, Y -15.360, Z 119.000}
   LaserStart_Ext()
   LIN {X -0.560, Y -15.360, Z 119.000}
   LaserEnd_Ext()
   LIN {X 10.998, Y -15.360, Z 119.000}
   LaserStart_Ext()
   LIN {X 13.327, Y -15.360, Z 119.000}
   LaserEnd_Ext()
   LIN {X 13.317, Y -14.360, Z 119.000}
   LaserStart_Ext()
   LIN {X 10.838, Y -14.360, Z 119.000}
   LaserEnd_Ext()
   LIN {X 0.003, Y -14.360, Z 119.000}
   LaserStart_Ext()
   LIN {X -2.378, Y -14.360, Z 119.000}
   LaserEnd_Ext()
   LIN {X -2.150, Y -13.360, Z 119.000}
   LaserStart_Ext()
   LIN {X 0.680, Y -13.360, Z 119.000}
   LaserEnd_Ext()
   LIN {X 10.277, Y -13.360, Z 119.000}
   LaserStart_Ext()
   LIN {X 13.303, Y -13.360, Z 119.000}
   LaserEnd_Ext()
   LIN {X 13.273, Y -12.360, Z 119.000}
   LaserStart_Ext()
   LIN {X 9.384, Y -12.360, Z 119.000}
   LaserEnd_Ext()
   LIN {X 1.309, Y -12.360, Z 119.000}
   LaserStart_Ext()
   LIN {X -1.928, Y -12.360, Z 119.000}
   LaserEnd_Ext()
   LIN {X -1.704, Y -11.360, Z 119.000}
   LaserStart_Ext()
   LIN {X 2.539, Y -11.360, Z 119.000}
   LaserEnd_Ext()
   LIN {X 8.138, Y -11.360, Z 119.000}
   LaserStart_Ext()
   LIN {X 13.236, Y -11.360, Z 119.000}
   LaserEnd_Ext()
   LIN {X 13.193, Y -10.360, Z 119.000}
   LaserStart_Ext()
   LIN {X -1.479, Y -10.360, Z 119.000}
   LaserEnd_Ext()
   LIN {X -1.254, Y -9.360, Z 119.000}
   LaserStart_Ext()
   LIN {X 13.139, Y -9.360, Z 119.000}
   LaserEnd_Ext()
   LIN {X 13.085, Y -8.360, Z 119.000}
   LaserStart_Ext()
   LIN {X -1.067, Y -8.360, Z 119.000}
   LaserEnd_Ext()
   LIN {X -0.920, Y -7.360, Z 119.000}
   LaserStart_Ext()
   LIN {X 12.993, Y -7.360, Z 119.000}
   LaserEnd_Ext()
   LIN {X 12.910, Y -6.360, Z 119.000}
   LaserStart_Ext()
   LIN {X -0.773, Y -6.360, Z 119.000}
   LaserEnd_Ext()
   LIN {X -0.626, Y -5.360, Z 119.000}
   LaserStart_Ext()
   LIN {X 12.829, Y -5.360, Z 119.000}
   LaserEnd_Ext()
   LIN {X 12.719, Y -4.360, Z 119.000}
   LaserStart_Ext()
   LIN {X -0.479, Y -4.360, Z 119.000}
   LaserEnd_Ext()
   LIN {X -0.373, Y -3.360, Z 119.000}
   LaserStart_Ext()
   LIN {X 12.598, Y -3.360, Z 119.000}
   LaserEnd_Ext()
   LIN {X 12.478, Y -2.360, Z 119.000}
   LaserStart_Ext()
   LIN {X -0.280, Y -2.360, Z 119.000}
   LaserEnd_Ext()
   LIN {X -0.212, Y -1.360, Z 119.000}
   LaserStart_Ext()
   LIN {X 12.347, Y -1.360, Z 119.000}
   LaserEnd_Ext()
   LIN {X 12.209, Y -0.360, Z 119.000}
   LaserStart_Ext()
   LIN {X -0.150, Y -0.360, Z 119.000}
   LaserEnd_Ext()
   LIN {X -0.088, Y 0.640, Z 119.000}
   LaserStart_Ext()
   LIN {X 12.070, Y 0.640, Z 119.000}
   LaserEnd_Ext()
   LIN {X 11.931, Y 1.640, Z 119.000}
   LaserStart_Ext()
   LIN {X -0.026, Y 1.640, Z 119.000}
   LaserEnd_Ext()
   LIN {X 0.009, Y 2.640, Z 119.000}
   LaserStart_Ext()
   LIN {X 11.754, Y 2.640, Z 119.000}
   LaserEnd_Ext()
   LIN {X 11.552, Y 3.640, Z 119.000}
   LaserStart_Ext()
   LIN {X -0.011, Y 3.640, Z 119.000}
   LaserEnd_Ext()
   LIN {X -0.031, Y 4.640, Z 119.000}
   LaserStart_Ext()
   LIN {X 11.351, Y 4.640, Z 119.000}
   LaserEnd_Ext()
   LIN {X 11.149, Y 5.640, Z 119.000}
   LaserStart_Ext()
   LIN {X -0.051, Y 5.640, Z 119.000}
   LaserEnd_Ext()
   LIN {X -0.071, Y 6.640, Z 119.000}
   LaserStart_Ext()
   LIN {X 10.947, Y 6.640, Z 119.000}
   LaserEnd_Ext()
   LIN {X 10.745, Y 7.640, Z 119.000}
   LaserStart_Ext()
   LIN {X -0.091, Y 7.640, Z 119.000}
   LaserEnd_Ext()
   LIN {X -0.112, Y 8.640, Z 119.000}
   LaserStart_Ext()
   LIN {X 10.539, Y 8.640, Z 119.000}
   LaserEnd_Ext()
   LIN {X 10.308, Y 9.640, Z 119.000}
   LaserStart_Ext()
   LIN {X -0.169, Y 9.640, Z 119.000}
   LaserEnd_Ext()
   LIN {X -0.236, Y 10.640, Z 119.000}
   LaserStart_Ext()
   LIN {X 10.077, Y 10.640, Z 119.000}
   LaserEnd_Ext()
   LIN {X 9.846, Y 11.640, Z 119.000}
   LaserStart_Ext()
   LIN {X -0.303, Y 11.640, Z 119.000}
   LaserEnd_Ext()
   LIN {X -0.424, Y 12.640, Z 119.000}
   LaserStart_Ext()
   LIN {X 9.576, Y 12.640, Z 119.000}
   LaserEnd_Ext()
   LIN {X 9.269, Y 13.640, Z 119.000}
   LaserStart_Ext()
   LIN {X -0.590, Y 13.640, Z 119.000}
   LaserEnd_Ext()
   LIN {X -0.756, Y 14.640, Z 119.000}
   LaserStart_Ext()
   LIN {X 8.962, Y 14.640, Z 119.000}
   LaserEnd_Ext()
   LIN {X 8.656, Y 15.640, Z 119.000}
   LaserStart_Ext()
   LIN {X -0.922, Y 15.640, Z 119.000}
   LaserEnd_Ext()
   LIN {X -1.089, Y 16.640, Z 119.000}
   LaserStart_Ext()
   LIN {X 8.349, Y 16.640, Z 119.000}
   LaserEnd_Ext()
   LIN {X 8.042, Y 17.640, Z 119.000}
   LaserStart_Ext()
   LIN {X -1.255, Y 17.640, Z 119.000}
   LaserEnd_Ext()
   LIN {X -1.421, Y 18.640, Z 119.000}
   LaserStart_Ext()
   LIN {X 7.736, Y 18.640, Z 119.000}
   LaserEnd_Ext()
   LIN {X 7.429, Y 19.640, Z 119.000}
   LaserStart_Ext()
   LIN {X -1.587, Y 19.640, Z 119.000}
   LaserEnd_Ext()
   LIN {X -1.770, Y 20.640, Z 119.000}
   LaserStart_Ext()
   LIN {X 7.106, Y 20.640, Z 119.000}
   LaserEnd_Ext()
   LIN {X 6.779, Y 21.640, Z 119.000}
   LaserStart_Ext()
   LIN {X -1.966, Y 21.640, Z 119.000}
   LaserEnd_Ext()
   LIN {X -2.206, Y 22.640, Z 119.000}
   LaserStart_Ext()
   LIN {X 6.389, Y 22.640, Z 119.000}
   LaserEnd_Ext()
   LIN {X 5.984, Y 23.640, Z 119.000}
   LaserStart_Ext()
   LIN {X -2.512, Y 23.640, Z 119.000}
   LaserEnd_Ext()
   LIN {X -2.819, Y 24.640, Z 119.000}
   LaserStart_Ext()
   LIN {X 5.579, Y 24.640, Z 119.000}
   LaserEnd_Ext()
   LIN {X 5.174, Y 25.640, Z 119.000}
   LaserStart_Ext()
   LIN {X -3.125, Y 25.640, Z 119.000}
   LaserEnd_Ext()
   LIN {X -3.432, Y 26.640, Z 119.000}
   LaserStart_Ext()
   LIN {X 4.768, Y 26.640, Z 119.000}
   LaserEnd_Ext()
   LIN {X 4.363, Y 27.640, Z 119.000}
   LaserStart_Ext()
   LIN {X -3.739, Y 27.640, Z 119.000}
   LaserEnd_Ext()
   LIN {X -4.045, Y 28.640, Z 119.000}
   LaserStart_Ext()
   LIN {X 3.959, Y 28.640, Z 119.000}
   LaserEnd_Ext()
   LIN {X 3.509, Y 29.640, Z 119.000}
   LaserStart_Ext()
   LIN {X -4.355, Y 29.640, Z 119.000}
   LaserEnd_Ext()
   LIN {X -4.722, Y 30.640, Z 119.000}
   LaserStart_Ext()
   LIN {X 3.025, Y 30.640, Z 119.000}
   LaserEnd_Ext()
   LIN {X 2.541, Y 31.640, Z 119.000}
   LaserStart_Ext()
   LIN {X -5.134, Y 31.640, Z 119.000}
   LaserEnd_Ext()
   LIN {X -5.550, Y 32.640, Z 119.000}
   LaserStart_Ext()
   LIN {X 2.057, Y 32.640, Z 119.000}
   LaserEnd_Ext()
   LIN {X 1.573, Y 33.640, Z 119.000}
   LaserStart_Ext()
   LIN {X -5.973, Y 33.640, Z 119.000}
   LaserEnd_Ext()
   LIN {X -6.397, Y 34.640, Z 119.000}
   LaserStart_Ext()
   LIN {X 1.080, Y 34.640, Z 119.000}
   LaserEnd_Ext()
   LIN {X 0.568, Y 35.640, Z 119.000}
   LaserStart_Ext()
   LIN {X -6.831, Y 35.640, Z 119.000}
   LaserEnd_Ext()
   LIN {X -7.311, Y 36.640, Z 119.000}
   LaserStart_Ext()
   LIN {X 0.021, Y 36.640, Z 119.000}
   LaserEnd_Ext()
   LIN {X -0.527, Y 37.640, Z 119.000}
   LaserStart_Ext()
   LIN {X -7.805, Y 37.640, Z 119.000}
   LaserEnd_Ext()
   LIN {X -8.300, Y 38.640, Z 119.000}
   LaserStart_Ext()
   LIN {X -1.080, Y 38.640, Z 119.000}
   LaserEnd_Ext()
   LIN {X -1.654, Y 39.640, Z 119.000}
   LaserStart_Ext()
   LIN {X -8.832, Y 39.640, Z 119.000}
   LaserEnd_Ext()
   LIN {X -9.387, Y 40.640, Z 119.000}
   LaserStart_Ext()
   LIN {X -2.249, Y 40.640, Z 119.000}
   LaserEnd_Ext()
   LIN {X -2.849, Y 41.640, Z 119.000}
   LaserStart_Ext()
   LIN {X -9.947, Y 41.640, Z 119.000}
   LaserEnd_Ext()
   LIN {X -10.387, Y 42.640, Z 119.000}
   LaserStart_Ext()
   LIN {X -3.468, Y 42.640, Z 119.000}
   LaserEnd_Ext()
   LIN {X -4.099, Y 43.640, Z 119.000}
   LaserStart_Ext()
   LIN {X -10.505, Y 43.640, Z 119.000}
   LaserEnd_Ext()
   LIN {X -10.366, Y 44.640, Z 119.000}
   LaserStart_Ext()
   LIN {X -4.746, Y 44.640, Z 119.000}
   LaserEnd_Ext()
   LIN {X -5.563, Y 45.640, Z 119.000}
   LaserStart_Ext()
   LIN {X -9.752, Y 45.640, Z 119.000}
   LaserEnd_Ext()
   LIN {X 1.364, Y -19.549, Z 119.850}
   LaserStart_Ext()
   LIN {X 0.668, Y -18.032, Z 119.850} C_DIS
   LIN {X 0.494, Y -17.584, Z 119.850} C_DIS
   LIN {X 0.454, Y -15.920, Z 119.850} C_DIS
   LIN {X 0.543, Y -15.418, Z 119.850} C_DIS
   LIN {X 1.841, Y -13.253, Z 119.850} C_DIS
   LIN {X 2.531, Y -12.438, Z 119.850} C_DIS
   LIN {X 4.036, Y -11.745, Z 119.850} C_DIS
   LIN {X 4.158, Y -11.688, Z 119.850} C_DIS
   LIN {X 4.288, Y -11.681, Z 119.850} C_DIS
   LIN {X 6.207, Y -11.579, Z 119.850} C_DIS
   LIN {X 7.807, Y -12.207, Z 119.850} C_DIS
   LIN {X 8.215, Y -12.374, Z 119.850} C_DIS
   LIN {X 8.427, Y -12.609, Z 119.850} C_DIS
   LIN {X 9.806, Y -14.142, Z 119.850} C_DIS
   LIN {X 10.131, Y -15.152, Z 119.850} C_DIS
   LIN {X 10.358, Y -16.816, Z 119.850} C_DIS
   LIN {X 10.250, Y -17.547, Z 119.850} C_DIS
   LIN {X 9.492, Y -19.330, Z 119.850} C_DIS
   LIN {X 9.202, Y -19.709, Z 119.850} C_DIS
   LIN {X 8.489, Y -20.444, Z 119.850} C_DIS
   LIN {X 7.004, Y -21.182, Z 119.850} C_DIS
   LIN {X 6.611, Y -21.380, Z 119.850} C_DIS
   LIN {X 5.942, Y -21.413, Z 119.850} C_DIS
   LIN {X 4.562, Y -21.484, Z 119.850} C_DIS
   LIN {X 3.670, Y -21.139, Z 119.850} C_DIS
   LIN {X 2.635, Y -20.736, Z 119.850} C_DIS
   LIN {X 1.859, Y -20.008, Z 119.850} C_DIS
   LIN {X 1.364, Y -19.549, Z 119.850}
   LaserEnd_Ext()
   LIN {X -3.377, Y -15.705, Z 119.850}
   LaserStart_Ext()
   LIN {X -3.323, Y -14.281, Z 119.850} C_DIS
   LIN {X -3.215, Y -13.808, Z 119.850} C_DIS
   LIN {X -2.160, Y -9.120, Z 119.850} C_DIS
   LIN {X -1.959, Y -7.943, Z 119.850} C_DIS
   LIN {X -1.445, Y -4.446, Z 119.850} C_DIS
   LIN {X -1.169, Y -1.471, Z 119.850} C_DIS
   LIN {X -0.961, Y 1.903, Z 119.850} C_DIS
   LIN {X -1.108, Y 9.255, Z 119.850} C_DIS
   LIN {X -1.261, Y 11.537, Z 119.850} C_DIS
   LIN {X -2.744, Y 20.471, Z 119.850} C_DIS
   LIN {X -3.005, Y 21.798, Z 119.850} C_DIS
   LIN {X -5.198, Y 28.951, Z 119.850} C_DIS
   LIN {X -5.431, Y 29.703, Z 119.850} C_DIS
   LIN {X -5.568, Y 30.023, Z 119.850} C_DIS
   LIN {X -6.862, Y 33.182, Z 119.850} C_DIS
   LIN {X -7.483, Y 34.650, Z 119.850} C_DIS
   LIN {X -8.666, Y 37.114, Z 119.850} C_DIS
   LIN {X -9.024, Y 37.837, Z 119.850} C_DIS
   LIN {X -10.036, Y 39.736, Z 119.850} C_DIS
   LIN {X -10.358, Y 40.311, Z 119.850} C_DIS
   LIN {X -11.091, Y 41.593, Z 119.850} C_DIS
   LIN {X -11.181, Y 41.835, Z 119.850} C_DIS
   LIN {X -11.594, Y 42.950, Z 119.850} C_DIS
   LIN {X -11.477, Y 44.692, Z 119.850} C_DIS
   LIN {X -11.467, Y 44.824, Z 119.850} C_DIS
   LIN {X -10.712, Y 46.095, Z 119.850} C_DIS
   LIN {X -2.555, Y 43.048, Z 119.850} C_DIS
   LIN {X -2.213, Y 42.505, Z 119.850} C_DIS
   LIN {X -0.431, Y 39.515, Z 119.850} C_DIS
   LIN {X -0.319, Y 39.318, Z 119.850} C_DIS
   LIN {X 1.802, Y 35.442, Z 119.850} C_DIS
   LIN {X 2.028, Y 34.988, Z 119.850} C_DIS
   LIN {X 4.742, Y 29.380, Z 119.850} C_DIS
   LIN {X 4.973, Y 28.807, Z 119.850} C_DIS
   LIN {X 7.757, Y 21.937, Z 119.850} C_DIS
   LIN {X 8.139, Y 20.770, Z 119.850} C_DIS
   LIN {X 10.878, Y 11.839, Z 119.850} C_DIS
   LIN {X 11.456, Y 9.336, Z 119.850} C_DIS
   LIN {X 12.990, Y 1.743, Z 119.850} C_DIS
   LIN {X 13.399, Y -1.209, Z 119.850} C_DIS
   LIN {X 13.902, Y -5.380, Z 119.850} C_DIS
   LIN {X 14.045, Y -7.132, Z 119.850} C_DIS
   LIN {X 14.108, Y -7.616, Z 119.850} C_DIS
   LIN {X 14.118, Y -7.766, Z 119.850} C_DIS
   LIN {X 14.337, Y -11.822, Z 119.850} C_DIS
   LIN {X 14.372, Y -12.766, Z 119.850} C_DIS
   LIN {X 14.418, Y -16.285, Z 119.850} C_DIS
   LIN {X 14.419, Y -16.516, Z 119.850} C_DIS
   LIN {X 14.360, Y -16.759, Z 119.850} C_DIS
   LIN {X 13.421, Y -20.581, Z 119.850} C_DIS
   LIN {X 13.112, Y -21.053, Z 119.850} C_DIS
   LIN {X 11.430, Y -23.138, Z 119.850} C_DIS
   LIN {X 10.892, Y -23.638, Z 119.850} C_DIS
   LIN {X 8.877, Y -24.640, Z 119.850} C_DIS
   LIN {X 7.281, Y -25.338, Z 119.850} C_DIS
   LIN {X 5.480, Y -25.418, Z 119.850} C_DIS
   LIN {X 3.741, Y -25.413, Z 119.850} C_DIS
   LIN {X 2.145, Y -24.835, Z 119.850} C_DIS
   LIN {X 0.521, Y -24.160, Z 119.850} C_DIS
   LIN {X -0.917, Y -22.786, Z 119.850} C_DIS
   LIN {X -2.209, Y -21.438, Z 119.850} C_DIS
   LIN {X -3.005, Y -19.445, Z 119.850} C_DIS
   LIN {X -3.517, Y -17.929, Z 119.850} C_DIS
   LIN {X -3.377, Y -15.705, Z 119.850}
   LaserEnd_Ext()
   LIN {X 12.602, Y -2.952, Z 119.850}
   LaserStart_Ext()
   LIN {X 12.602, Y -19.725, Z 119.850}
   LaserEnd_Ext()
   LIN {X 11.602, Y -21.332, Z 119.850}
   LaserStart_Ext()
   LIN {X 11.602, Y 3.562, Z 119.850}
   LaserEnd_Ext()
   LIN {X 10.602, Y 8.515, Z 119.850}
   LaserStart_Ext()
   LIN {X 10.602, Y -13.537, Z 119.850}
   LaserEnd_Ext()
   LIN {X 10.602, Y -19.276, Z 119.850}
   LaserStart_Ext()
   LIN {X 10.602, Y -22.542, Z 119.850}
   LaserEnd_Ext()
   LIN {X 9.602, Y -23.163, Z 119.850}
   LaserStart_Ext()
   LIN {X 9.602, Y -20.733, Z 119.850}
   LaserEnd_Ext()
   LIN {X 9.602, Y -12.420, Z 119.850}
   LaserStart_Ext()
   LIN {X 9.602, Y 12.590, Z 119.850}
   LaserEnd_Ext()
   LIN {X 8.602, Y 15.851, Z 119.850}
   LaserStart_Ext()
   LIN {X 8.602, Y -11.453, Z 119.850}
   LaserEnd_Ext()
   LIN {X 8.602, Y -21.505, Z 119.850}
   LaserStart_Ext()
   LIN {X 8.602, Y -23.660, Z 119.850}
   LaserEnd_Ext()
   LIN {X 7.602, Y -24.106, Z 119.850}
   LaserStart_Ext()
   LIN {X 7.602, Y -22.002, Z 119.850}
   LaserEnd_Ext()
   LIN {X 7.602, Y -11.053, Z 119.850}
   LaserStart_Ext()
   LIN {X 7.602, Y 19.112, Z 119.850}
   LaserEnd_Ext()
   LIN {X 6.602, Y 22.126, Z 119.850}
   LaserStart_Ext()
   LIN {X 6.602, Y -10.660, Z 119.850}
   LaserEnd_Ext()
   LIN {X 6.602, Y -22.382, Z 119.850}
   LaserStart_Ext()
   LIN {X 6.602, Y -24.367, Z 119.850}
   LaserEnd_Ext()
   LIN {X 5.602, Y -24.412, Z 119.850}
   LaserStart_Ext()
   LIN {X 5.602, Y -22.431, Z 119.850}
   LaserEnd_Ext()
   LIN {X 5.602, Y -10.610, Z 119.850}
   LaserStart_Ext()
   LIN {X 5.602, Y 24.594, Z 119.850}
   LaserEnd_Ext()
   LIN {X 4.602, Y 27.061, Z 119.850}
   LaserStart_Ext()
   LIN {X 4.602, Y -10.663, Z 119.850}
   LaserEnd_Ext()
   LIN {X 4.602, Y -22.482, Z 119.850}
   LaserStart_Ext()
   LIN {X 4.602, Y -24.416, Z 119.850}
   LaserEnd_Ext()
   LIN {X 3.602, Y -24.299, Z 119.850}
   LaserStart_Ext()
   LIN {X 3.602, Y -22.185, Z 119.850}
   LaserEnd_Ext()
   LIN {X 3.602, Y -10.844, Z 119.850}
   LaserStart_Ext()
   LIN {X 3.602, Y 29.441, Z 119.850}
   LaserEnd_Ext()
   LIN {X 2.602, Y 31.507, Z 119.850}
   LaserStart_Ext()
   LIN {X 2.602, Y -11.304, Z 119.850}
   LaserEnd_Ext()
   LIN {X 2.602, Y -21.796, Z 119.850}
   LaserStart_Ext()
   LIN {X 2.602, Y -23.937, Z 119.850}
   LaserEnd_Ext()
   LIN {X 1.602, Y -23.526, Z 119.850}
   LaserStart_Ext()
   LIN {X 1.602, Y -21.138, Z 119.850}
   LaserEnd_Ext()
   LIN {X 1.602, Y -11.988, Z 119.850}
   LaserStart_Ext()
   LIN {X 1.602, Y 33.574, Z 119.850}
   LaserEnd_Ext()
   LIN {X 0.602, Y 35.552, Z 119.850}
   LaserStart_Ext()
   LIN {X 0.602, Y -13.375, Z 119.850}
   LaserEnd_Ext()
   LIN {X 0.602, Y -20.195, Z 119.850}
   LaserStart_Ext()
   LIN {X 0.602, Y -22.854, Z 119.850}
   LaserEnd_Ext()
   LIN {X -0.398, Y -21.882, Z 119.850}
   LaserStart_Ext()
   LIN {X -0.398, Y -18.049, Z 119.850}
   LaserEnd_Ext()
   LIN {X -0.398, Y -15.080, Z 119.850}
   LaserStart_Ext()
   LIN {X -0.398, Y -3.987, Z 119.850}
   LaserEnd_Ext()
   LIN {X -0.398, Y 12.447, Z 119.850}
   LaserStart_Ext()
   LIN {X -0.398, Y 37.379, Z 119.850}
   LaserEnd_Ext()
   LIN {X -1.398, Y 39.184, Z 119.850}
   LaserStart_Ext()
   LIN {X -1.398, Y 18.468, Z 119.850}
   LaserEnd_Ext()
   LIN {X -1.398, Y -10.291, Z 119.850}
   LaserStart_Ext()
   LIN {X -1.398, Y -20.771, Z 119.850}
   LaserEnd_Ext()
   LIN {X -2.398, Y -18.117, Z 119.850}
   LaserStart_Ext()
   LIN {X -2.398, Y -16.076, Z 119.850}
   LaserEnd_Ext()
   LIN {X -2.398, Y 23.230, Z 119.850}
   LaserStart_Ext()
   LIN {X -2.398, Y 40.864, Z 119.850}
   LaserEnd_Ext()
   LIN {X -3.398, Y 42.295, Z 119.850}
   LaserStart_Ext()
   LIN {X -3.398, Y 26.492, Z 119.850}
   LaserEnd_Ext()
   LIN {X -4.398, Y 29.748, Z 119.850}
   LaserStart_Ext()
   LIN {X -4.398, Y 42.669, Z 119.850}
   LaserEnd_Ext()
   LIN {X -5.398, Y 43.042, Z 119.850}
   LaserStart_Ext()
   LIN {X -5.398, Y 32.247, Z 119.850}
   LaserEnd_Ext()
   LIN {X -6.398, Y 34.653, Z 119.850}
   LaserStart_Ext()
   LIN {X -6.398, Y 43.416, Z 119.850}
   LaserEnd_Ext()
   LIN {X -7.398, Y 43.789, Z 119.850}
   LaserStart_Ext()
   LIN {X -7.398, Y 36.784, Z 119.850}
   LaserEnd_Ext()
   LIN {X -8.398, Y 38.789, Z 119.850}
   LaserStart_Ext()
   LIN {X -8.398, Y 44.163, Z 119.850}
   LaserEnd_Ext()
   LIN {X -9.398, Y 44.536, Z 119.850}
   LaserStart_Ext()
   LIN {X -9.398, Y 40.644, Z 119.850}
   LaserEnd_Ext()
   LIN {X -10.398, Y 42.600, Z 119.850}
   LaserStart_Ext()
   LIN {X -10.398, Y 44.666, Z 119.850}
   LaserEnd_Ext()
   LIN {X 4.125, Y -11.661, Z 120.700}
   LaserStart_Ext()
   LIN {X 5.770, Y -11.542, Z 120.700} C_DIS
   LIN {X 6.280, Y -11.515, Z 120.700} C_DIS
   LIN {X 6.649, Y -11.659, Z 120.700} C_DIS
   LIN {X 8.376, Y -12.366, Z 120.700} C_DIS
   LIN {X 9.274, Y -13.360, Z 120.700} C_DIS
   LIN {X 9.850, Y -14.001, Z 120.700} C_DIS
   LIN {X 10.362, Y -15.590, Z 120.700} C_DIS
   LIN {X 10.450, Y -16.238, Z 120.700} C_DIS
   LIN {X 10.192, Y -17.992, Z 120.700} C_DIS
   LIN {X 9.846, Y -18.806, Z 120.700} C_DIS
   LIN {X 8.909, Y -20.028, Z 120.700} C_DIS
   LIN {X 8.534, Y -20.414, Z 120.700} C_DIS
   LIN {X 7.366, Y -20.994, Z 120.700} C_DIS
   LIN {X 5.895, Y -21.359, Z 120.700} C_DIS
   LIN {X 4.660, Y -21.423, Z 120.700} C_DIS
   LIN {X 3.018, Y -20.789, Z 120.700} C_DIS
   LIN {X 2.715, Y -20.668, Z 120.700} C_DIS
   LIN {X 2.572, Y -20.531, Z 120.700} C_DIS
   LIN {X 1.457, Y -19.496, Z 120.700} C_DIS
   LIN {X 1.080, Y -18.674, Z 120.700} C_DIS
   LIN {X 0.538, Y -17.280, Z 120.700} C_DIS
   LIN {X 0.518, Y -16.418, Z 120.700} C_DIS
   LIN {X 0.799, Y -14.826, Z 120.700} C_DIS
   LIN {X 1.397, Y -13.829, Z 120.700} C_DIS
   LIN {X 2.643, Y -12.356, Z 120.700} C_DIS
   LIN {X 3.322, Y -12.044, Z 120.700} C_DIS
   LIN {X 4.125, Y -11.661, Z 120.700}
   LaserEnd_Ext()
   LIN {X 14.439, Y -12.488, Z 120.700}
   LaserStart_Ext()
   LIN {X 14.224, Y -8.455, Z 120.700} C_DIS
   LIN {X 14.155, Y -7.403, Z 120.700} C_DIS
   LIN {X 14.104, Y -7.018, Z 120.700} C_DIS
   LIN {X 14.003, Y -5.779, Z 120.700} C_DIS
   LIN {X 13.383, Y -0.643, Z 120.700} C_DIS
   LIN {X 13.116, Y 1.284, Z 120.700} C_DIS
   LIN {X 11.363, Y 9.964, Z 120.700} C_DIS
   LIN {X 11.056, Y 11.295, Z 120.700} C_DIS
   LIN {X 7.966, Y 21.373, Z 120.700} C_DIS
   LIN {X 7.861, Y 21.693, Z 120.700} C_DIS
   LIN {X 5.601, Y 27.270, Z 120.700} C_DIS
   LIN {X -6.271, Y 31.702, Z 120.700} C_DIS
   LIN {X -5.424, Y 29.633, Z 120.700} C_DIS
   LIN {X -5.378, Y 29.500, Z 120.700} C_DIS
   LIN {X -2.953, Y 21.591, Z 120.700} C_DIS
   LIN {X -2.845, Y 21.041, Z 120.700} C_DIS
   LIN {X -1.194, Y 11.100, Z 120.700} C_DIS
   LIN {X -1.102, Y 9.724, Z 120.700} C_DIS
   LIN {X -0.936, Y 1.465, Z 120.700} C_DIS
   LIN {X -1.081, Y -0.886, Z 120.700} C_DIS
   LIN {X -1.452, Y -4.885, Z 120.700} C_DIS
   LIN {X -1.832, Y -7.470, Z 120.700} C_DIS
   LIN {X -2.173, Y -9.468, Z 120.700} C_DIS
   LIN {X -2.977, Y -13.040, Z 120.700} C_DIS
   LIN {X -3.251, Y -14.238, Z 120.700} C_DIS
   LIN {X -3.387, Y -17.846, Z 120.700} C_DIS
   LIN {X -3.402, Y -18.076, Z 120.700} C_DIS
   LIN {X -3.349, Y -18.232, Z 120.700} C_DIS
   LIN {X -2.046, Y -21.494, Z 120.700} C_DIS
   LIN {X -1.716, Y -21.839, Z 120.700} C_DIS
   LIN {X 0.728, Y -24.173, Z 120.700} C_DIS
   LIN {X 1.248, Y -24.389, Z 120.700} C_DIS
   LIN {X 3.968, Y -25.376, Z 120.700} C_DIS
   LIN {X 4.523, Y -25.378, Z 120.700} C_DIS
   LIN {X 7.508, Y -25.245, Z 120.700} C_DIS
   LIN {X 7.926, Y -25.062, Z 120.700} C_DIS
   LIN {X 11.094, Y -23.487, Z 120.700} C_DIS
   LIN {X 12.027, Y -22.348, Z 120.700} C_DIS
   LIN {X 13.410, Y -20.657, Z 120.700} C_DIS
   LIN {X 13.510, Y -20.508, Z 120.700} C_DIS
   LIN {X 14.366, Y -17.097, Z 120.700} C_DIS
   LIN {X 14.496, Y -16.435, Z 120.700} C_DIS
   LIN {X 14.450, Y -12.942, Z 120.700} C_DIS
   LIN {X 14.439, Y -12.488, Z 120.700}
   LaserEnd_Ext()
   LIN {X -4.338, Y 29.522, Z 120.700}
   LaserStart_Ext()
   LIN {X -3.290, Y 29.522, Z 120.700}
   LaserEnd_Ext()
   LIN {X -0.611, Y 28.522, Z 120.700}
   LaserStart_Ext()
   LIN {X -4.032, Y 28.522, Z 120.700}
   LaserEnd_Ext()
   LIN {X -3.725, Y 27.522, Z 120.700}
   LaserStart_Ext()
   LIN {X 2.067, Y 27.522, Z 120.700}
   LaserEnd_Ext()
   LIN {X 4.746, Y 26.522, Z 120.700}
   LaserStart_Ext()
   LIN {X -3.419, Y 26.522, Z 120.700}
   LaserEnd_Ext()
   LIN {X -3.112, Y 25.522, Z 120.700}
   LaserStart_Ext()
   LIN {X 5.230, Y 25.522, Z 120.700}
   LaserEnd_Ext()
   LIN {X 5.635, Y 24.522, Z 120.700}
   LaserStart_Ext()
   LIN {X -2.806, Y 24.522, Z 120.700}
   LaserEnd_Ext()
   LIN {X -2.499, Y 23.522, Z 120.700}
   LaserStart_Ext()
   LIN {X 6.041, Y 23.522, Z 120.700}
   LaserEnd_Ext()
   LIN {X 6.446, Y 22.522, Z 120.700}
   LaserStart_Ext()
   LIN {X -2.192, Y 22.522, Z 120.700}
   LaserEnd_Ext()
   LIN {X -1.920, Y 21.522, Z 120.700}
   LaserStart_Ext()
   LIN {X 6.851, Y 21.522, Z 120.700}
   LaserEnd_Ext()
   LIN {X 7.181, Y 20.522, Z 120.700}
   LaserStart_Ext()
   LIN {X -1.745, Y 20.522, Z 120.700}
   LaserEnd_Ext()
   LIN {X -1.579, Y 19.522, Z 120.700}
   LaserStart_Ext()
   LIN {X 7.487, Y 19.522, Z 120.700}
   LaserEnd_Ext()
   LIN {X 7.794, Y 18.522, Z 120.700}
   LaserStart_Ext()
   LIN {X -1.413, Y 18.522, Z 120.700}
   LaserEnd_Ext()
   LIN {X -1.247, Y 17.522, Z 120.700}
   LaserStart_Ext()
   LIN {X 8.101, Y 17.522, Z 120.700}
   LaserEnd_Ext()
   LIN {X 8.407, Y 16.522, Z 120.700}
   LaserStart_Ext()
   LIN {X -1.081, Y 16.522, Z 120.700}
   LaserEnd_Ext()
   LIN {X -0.915, Y 15.522, Z 120.700}
   LaserStart_Ext()
   LIN {X 8.714, Y 15.522, Z 120.700}
   LaserEnd_Ext()
   LIN {X 9.020, Y 14.522, Z 120.700}
   LaserStart_Ext()
   LIN {X -0.748, Y 14.522, Z 120.700}
   LaserEnd_Ext()
   LIN {X -0.582, Y 13.522, Z 120.700}
   LaserStart_Ext()
   LIN {X 9.327, Y 13.522, Z 120.700}
   LaserEnd_Ext()
   LIN {X 9.634, Y 12.522, Z 120.700}
   LaserStart_Ext()
   LIN {X -0.416, Y 12.522, Z 120.700}
   LaserEnd_Ext()
   LIN {X -0.250, Y 11.522, Z 120.700}
   LaserStart_Ext()
   LIN {X 9.940, Y 11.522, Z 120.700}
   LaserEnd_Ext()
   LIN {X 10.208, Y 10.522, Z 120.700}
   LaserStart_Ext()
   LIN {X -0.153, Y 10.522, Z 120.700}
   LaserEnd_Ext()
   LIN {X -0.098, Y 9.522, Z 120.700}
   LaserStart_Ext()
   LIN {X 10.432, Y 9.522, Z 120.700}
   LaserEnd_Ext()
   LIN {X 10.634, Y 8.522, Z 120.700}
   LaserStart_Ext()
   LIN {X -0.078, Y 8.522, Z 120.700}
   LaserEnd_Ext()
   LIN {X -0.058, Y 7.522, Z 120.700}
   LaserStart_Ext()
   LIN {X 10.836, Y 7.522, Z 120.700}
   LaserEnd_Ext()
   LIN {X 11.038, Y 6.522, Z 120.700}
   LaserStart_Ext()
   LIN {X -0.037, Y 6.522, Z 120.700}
   LaserEnd_Ext()
   LIN {X -0.017, Y 5.522, Z 120.700}
   LaserStart_Ext()
   LIN {X 11.240, Y 5.522, Z 120.700}
   LaserEnd_Ext()
   LIN {X 11.442, Y 4.522, Z 120.700}
   LaserStart_Ext()
   LIN {X 0.003, Y 4.522, Z 120.700}
   LaserEnd_Ext()
   LIN {X 0.023, Y 3.522, Z 120.700}
   LaserStart_Ext()
   LIN {X 11.644, Y 3.522, Z 120.700}
   LaserEnd_Ext()
   LIN {X 11.846, Y 2.522, Z 120.700}
   LaserStart_Ext()
   LIN {X 0.043, Y 2.522, Z 120.700}
   LaserEnd_Ext()
   LIN {X 0.063, Y 1.522, Z 120.700}
   LaserStart_Ext()
   LIN {X 12.048, Y 1.522, Z 120.700}
   LaserEnd_Ext()
   LIN {X 12.212, Y 0.522, Z 120.700}
   LaserStart_Ext()
   LIN {X 0.008, Y 0.522, Z 120.700}
   LaserEnd_Ext()
   LIN {X -0.054, Y -0.478, Z 120.700}
   LaserStart_Ext()
   LIN {X 12.351, Y -0.478, Z 120.700}
   LaserEnd_Ext()
   LIN {X 12.477, Y -1.478, Z 120.700}
   LaserStart_Ext()
   LIN {X -0.132, Y -1.478, Z 120.700}
   LaserEnd_Ext()
   LIN {X -0.225, Y -2.478, Z 120.700}
   LaserStart_Ext()
   LIN {X 12.597, Y -2.478, Z 120.700}
   LaserEnd_Ext()
   LIN {X 12.718, Y -3.478, Z 120.700}
   LaserStart_Ext()
   LIN {X -0.318, Y -3.478, Z 120.700}
   LaserEnd_Ext()
   LIN {X -0.410, Y -4.478, Z 120.700}
   LaserStart_Ext()
   LIN {X 12.839, Y -4.478, Z 120.700}
   LaserEnd_Ext()
   LIN {X 12.960, Y -5.478, Z 120.700}
   LaserStart_Ext()
   LIN {X -0.529, Y -5.478, Z 120.700}
   LaserEnd_Ext()
   LIN {X -0.676, Y -6.478, Z 120.700}
   LaserStart_Ext()
   LIN {X 13.057, Y -6.478, Z 120.700}
   LaserEnd_Ext()
   LIN {X 13.156, Y -7.478, Z 120.700}
   LaserStart_Ext()
   LIN {X -0.823, Y -7.478, Z 120.700}
   LaserEnd_Ext()
   LIN {X -0.990, Y -8.478, Z 120.700}
   LaserStart_Ext()
   LIN {X 13.224, Y -8.478, Z 120.700}
   LaserEnd_Ext()
   LIN {X 13.277, Y -9.478, Z 120.700}
   LaserStart_Ext()
   LIN {X -1.160, Y -9.478, Z 120.700}
   LaserEnd_Ext()
   LIN {X -1.375, Y -10.478, Z 120.700}
   LaserStart_Ext()
   LIN {X 13.331, Y -10.478, Z 120.700}
   LaserEnd_Ext()
   LIN {X 13.384, Y -11.478, Z 120.700}
   LaserStart_Ext()
   LIN {X 8.836, Y -11.478, Z 120.700}
   LaserEnd_Ext()
   LIN {X 2.167, Y -11.478, Z 120.700}
   LaserStart_Ext()
   LIN {X -1.600, Y -11.478, Z 120.700}
   LaserEnd_Ext()
   LIN {X -1.825, Y -12.478, Z 120.700}
   LaserStart_Ext()
   LIN {X 1.230, Y -12.478, Z 120.700}
   LaserEnd_Ext()
   LIN {X 9.825, Y -12.478, Z 120.700}
   LaserStart_Ext()
   LIN {X 13.437, Y -12.478, Z 120.700}
   LaserEnd_Ext()
   LIN {X 13.457, Y -13.478, Z 120.700}
   LaserStart_Ext()
   LIN {X 10.702, Y -13.478, Z 120.700}
   LaserEnd_Ext()
   LIN {X 0.441, Y -13.478, Z 120.700}
   LaserStart_Ext()
   LIN {X -2.051, Y -13.478, Z 120.700}
   LaserEnd_Ext()
   LIN {X -2.259, Y -14.478, Z 120.700}
   LaserStart_Ext()
   LIN {X -0.139, Y -14.478, Z 120.700}
   LaserEnd_Ext()
   LIN {X 11.054, Y -14.478, Z 120.700}
   LaserStart_Ext()
   LIN {X 13.470, Y -14.478, Z 120.700}
   LaserEnd_Ext()
   LIN {X 13.483, Y -15.478, Z 120.700}
   LaserStart_Ext()
   LIN {X 11.356, Y -15.478, Z 120.700}
   LaserEnd_Ext()
   LIN {X -0.332, Y -15.478, Z 120.700}
   LaserStart_Ext()
   LIN {X -2.297, Y -15.478, Z 120.700}
   LaserEnd_Ext()
   LIN {X -2.335, Y -16.478, Z 120.700}
   LaserStart_Ext()
   LIN {X -0.481, Y -16.478, Z 120.700}
   LaserEnd_Ext()
   LIN {X 11.425, Y -16.478, Z 120.700}
   LaserStart_Ext()
   LIN {X 13.468, Y -16.478, Z 120.700}
   LaserEnd_Ext()
   LIN {X 13.239, Y -17.478, Z 120.700}
   LaserStart_Ext()
   LIN {X 11.278, Y -17.478, Z 120.700}
   LaserEnd_Ext()
   LIN {X -0.442, Y -17.478, Z 120.700}
   LaserStart_Ext()
   LIN {X -2.373, Y -17.478, Z 120.700}
   LaserEnd_Ext()
   LIN {X -2.174, Y -18.478, Z 120.700}
   LaserStart_Ext()
   LIN {X -0.069, Y -18.478, Z 120.700}
   LaserEnd_Ext()
   LIN {X 11.072, Y -18.478, Z 120.700}
   LaserStart_Ext()
   LIN {X 12.988, Y -18.478, Z 120.700}
   LaserEnd_Ext()
   LIN {X 12.738, Y -19.478, Z 120.700}
   LaserStart_Ext()
   LIN {X 10.591, Y -19.478, Z 120.700}
   LaserEnd_Ext()
   LIN {X 0.348, Y -19.478, Z 120.700}
   LaserStart_Ext()
   LIN {X -1.774, Y -19.478, Z 120.700}
   LaserEnd_Ext()
   LIN {X -1.375, Y -20.478, Z 120.700}
   LaserStart_Ext()
   LIN {X 1.045, Y -20.478, Z 120.700}
   LaserEnd_Ext()
   LIN {X 9.823, Y -20.478, Z 120.700}
   LaserStart_Ext()
   LIN {X 12.264, Y -20.478, Z 120.700}
   LaserEnd_Ext()
   LIN {X 11.446, Y -21.478, Z 120.700}
   LaserStart_Ext()
   LIN {X 8.639, Y -21.478, Z 120.700}
   LaserEnd_Ext()
   LIN {X 2.131, Y -21.478, Z 120.700}
   LaserStart_Ext()
   LIN {X -0.645, Y -21.478, Z 120.700}
   LaserEnd_Ext()
   LIN {X 0.401, Y -22.478, Z 120.700}
   LaserStart_Ext()
   LIN {X 10.637, Y -22.478, Z 120.700}
   LaserEnd_Ext()
   LIN {X 8.865, Y -23.478, Z 120.700}
   LaserStart_Ext()
   LIN {X 1.669, Y -23.478, Z 120.700}
   LaserEnd_Ext()
   LIN {X 9.753, Y -13.709, Z 121.550}
   LaserStart_Ext()
   LIN {X 9.941, Y -13.967, Z 121.550} C_DIS
   LIN {X 10.492, Y -15.668, Z 121.550} C_DIS
   LIN {X 10.530, Y -16.024, Z 121.550} C_DIS
   LIN {X 10.177, Y -18.279, Z 121.550} C_DIS
   LIN {X 10.113, Y -18.426, Z 121.550} C_DIS
   LIN {X 9.207, Y -19.576, Z 121.550} C_DIS
   LIN {X 8.616, Y -20.346, Z 121.550} C_DIS
   LIN {X 8.468, Y -20.439, Z 121.550} C_DIS
   LIN {X 5.114, Y -21.271, Z 121.550} C_DIS
   LIN {X 4.769, Y -21.361, Z 121.550} C_DIS
   LIN {X 2.698, Y -20.540, Z 121.550} C_DIS
   LIN {X 1.721, Y -19.602, Z 121.550} C_DIS
   LIN {X 1.549, Y -19.443, Z 121.550} C_DIS
   LIN {X 1.491, Y -19.317, Z 121.550} C_DIS
   LIN {X 0.583, Y -16.977, Z 121.550} C_DIS
   LIN {X 0.735, Y -16.046, Z 121.550} C_DIS
   LIN {X 1.005, Y -14.386, Z 121.550} C_DIS
   LIN {X 1.068, Y -14.248, Z 121.550} C_DIS
   LIN {X 2.599, Y -12.413, Z 121.550} C_DIS
   LIN {X 2.897, Y -12.201, Z 121.550} C_DIS
   LIN {X 4.075, Y -11.639, Z 121.550} C_DIS
   LIN {X 5.719, Y -11.520, Z 121.550} C_DIS
   LIN {X 6.346, Y -11.451, Z 121.550} C_DIS
   LIN {X 8.373, Y -12.289, Z 121.550} C_DIS
   LIN {X 8.535, Y -12.359, Z 121.550} C_DIS
   LIN {X 9.753, Y -13.709, Z 121.550}
   LaserEnd_Ext()
   LIN {X 0.518, Y -23.844, Z 121.550}
   LaserStart_Ext()
   LIN {X 0.961, Y -24.200, Z 121.550} C_DIS
   LIN {X 3.743, Y -25.209, Z 121.550} C_DIS
   LIN {X 4.225, Y -25.338, Z 121.550} C_DIS
   LIN {X 7.166, Y -25.213, Z 121.550} C_DIS
   LIN {X 7.768, Y -25.134, Z 121.550} C_DIS
   LIN {X 10.543, Y -23.767, Z 121.550} C_DIS
   LIN {X 11.324, Y -23.291, Z 121.550} C_DIS
   LIN {X 13.023, Y -21.213, Z 121.550} C_DIS
   LIN {X 13.673, Y -20.253, Z 121.550} C_DIS
   LIN {X 14.280, Y -17.835, Z 121.550} C_DIS
   LIN {X 14.569, Y -16.355, Z 121.550} C_DIS
   LIN {X 14.539, Y -13.973, Z 121.550} C_DIS
   LIN {X 14.496, Y -12.214, Z 121.550} C_DIS
   LIN {X 14.358, Y -9.621, Z 121.550} C_DIS
   LIN {X 14.193, Y -7.130, Z 121.550} C_DIS
   LIN {X 14.163, Y -6.905, Z 121.550} C_DIS
   LIN {X 14.104, Y -6.178, Z 121.550} C_DIS
   LIN {X 13.367, Y -0.077, Z 121.550} C_DIS
   LIN {X 13.242, Y 0.826, Z 121.550} C_DIS
   LIN {X 11.271, Y 10.591, Z 121.550} C_DIS
   LIN {X 11.233, Y 10.752, Z 121.550} C_DIS
   LIN {X 10.650, Y 12.653, Z 121.550} C_DIS
   LIN {X -2.258, Y 17.471, Z 121.550} C_DIS
   LIN {X -1.127, Y 10.663, Z 121.550} C_DIS
   LIN {X -1.096, Y 10.193, Z 121.550} C_DIS
   LIN {X -0.911, Y 1.027, Z 121.550} C_DIS
   LIN {X -0.993, Y -0.300, Z 121.550} C_DIS
   LIN {X -1.460, Y -5.325, Z 121.550} C_DIS
   LIN {X -1.706, Y -6.996, Z 121.550} C_DIS
   LIN {X -2.186, Y -9.815, Z 121.550} C_DIS
   LIN {X -2.739, Y -12.272, Z 121.550} C_DIS
   LIN {X -3.179, Y -14.194, Z 121.550} C_DIS
   LIN {X -3.287, Y -17.045, Z 121.550} C_DIS
   LIN {X -3.285, Y -18.216, Z 121.550} C_DIS
   LIN {X -2.169, Y -20.971, Z 121.550} C_DIS
   LIN {X -1.861, Y -21.583, Z 121.550} C_DIS
   LIN {X 0.518, Y -23.844, Z 121.550}
   LaserEnd_Ext()
   LIN {X -2.280, Y -16.877, Z 121.550}
   LaserStart_Ext()
   LIN {X -2.280, Y -18.033, Z 121.550}
   LaserEnd_Ext()
   LIN {X -1.280, Y -20.503, Z 121.550}
   LaserStart_Ext()
   LIN {X -1.280, Y -10.342, Z 121.550}
   LaserEnd_Ext()
   LIN {X -0.280, Y 15.665, Z 121.550}
   LaserStart_Ext()
   LIN {X -0.280, Y 11.665, Z 121.550}
   LaserEnd_Ext()
   LIN {X -0.280, Y -3.432, Z 121.550}
   LaserStart_Ext()
   LIN {X -0.280, Y -16.041, Z 121.550}
   LaserEnd_Ext()
   LIN {X -0.280, Y -17.518, Z 121.550}
   LaserStart_Ext()
   LIN {X -0.280, Y -21.706, Z 121.550}
   LaserEnd_Ext()
   LIN {X 0.720, Y -22.657, Z 121.550}
   LaserStart_Ext()
   LIN {X 0.720, Y -20.001, Z 121.550}
   LaserEnd_Ext()
   LIN {X 0.720, Y -13.103, Z 121.550}
   LaserStart_Ext()
   LIN {X 0.720, Y 15.291, Z 121.550}
   LaserEnd_Ext()
   LIN {X 1.720, Y 14.918, Z 121.550}
   LaserStart_Ext()
   LIN {X 1.720, Y -11.905, Z 121.550}
   LaserEnd_Ext()
   LIN {X 1.720, Y -20.988, Z 121.550}
   LaserStart_Ext()
   LIN {X 1.720, Y -23.412, Z 121.550}
   LaserEnd_Ext()
   LIN {X 2.720, Y -23.774, Z 121.550}
   LaserStart_Ext()
   LIN {X 2.720, Y -21.626, Z 121.550}
   LaserEnd_Ext()
   LIN {X 2.720, Y -11.177, Z 121.550}
   LaserStart_Ext()
   LIN {X 2.720, Y 14.545, Z 121.550}
   LaserEnd_Ext()
   LIN {X 3.720, Y 14.172, Z 121.550}
   LaserStart_Ext()
   LIN {X 3.720, Y -10.704, Z 121.550}
   LaserEnd_Ext()
   LIN {X 3.720, Y -22.024, Z 121.550}
   LaserStart_Ext()
   LIN {X 3.720, Y -24.137, Z 121.550}
   LaserEnd_Ext()
   LIN {X 4.720, Y -24.316, Z 121.550}
   LaserStart_Ext()
   LIN {X 4.720, Y -22.360, Z 121.550}
   LaserEnd_Ext()
   LIN {X 4.720, Y -10.589, Z 121.550}
   LaserStart_Ext()
   LIN {X 4.720, Y 13.799, Z 121.550}
   LaserEnd_Ext()
   LIN {X 5.720, Y 13.425, Z 121.550}
   LaserStart_Ext()
   LIN {X 5.720, Y -10.514, Z 121.550}
   LaserEnd_Ext()
   LIN {X 5.720, Y -22.151, Z 121.550}
   LaserStart_Ext()
   LIN {X 5.720, Y -24.273, Z 121.550}
   LaserEnd_Ext()
   LIN {X 6.720, Y -24.231, Z 121.550}
   LaserStart_Ext()
   LIN {X 6.720, Y -21.903, Z 121.550}
   LaserEnd_Ext()
   LIN {X 6.720, Y -10.524, Z 121.550}
   LaserStart_Ext()
   LIN {X 6.720, Y 13.052, Z 121.550}
   LaserEnd_Ext()
   LIN {X 7.720, Y 12.679, Z 121.550}
   LaserStart_Ext()
   LIN {X 7.720, Y -10.937, Z 121.550}
   LaserEnd_Ext()
   LIN {X 7.720, Y -21.655, Z 121.550}
   LaserStart_Ext()
   LIN {X 7.720, Y -24.042, Z 121.550}
   LaserEnd_Ext()
   LIN {X 8.720, Y -23.550, Z 121.550}
   LaserStart_Ext()
   LIN {X 8.720, Y -21.406, Z 121.550}
   LaserEnd_Ext()
   LIN {X 8.720, Y -11.350, Z 121.550}
   LaserStart_Ext()
   LIN {X 8.720, Y 12.306, Z 121.550}
   LaserEnd_Ext()
   LIN {X 9.720, Y 11.933, Z 121.550}
   LaserStart_Ext()
   LIN {X 9.720, Y -12.180, Z 121.550}
   LaserEnd_Ext()
   LIN {X 9.720, Y -20.550, Z 121.550}
   LaserStart_Ext()
   LIN {X 9.720, Y -23.057, Z 121.550}
   LaserEnd_Ext()
   LIN {X 10.720, Y -22.449, Z 121.550}
   LaserStart_Ext()
   LIN {X 10.720, Y -19.271, Z 121.550}
   LaserEnd_Ext()
   LIN {X 10.720, Y -13.337, Z 121.550}
   LaserStart_Ext()
   LIN {X 10.720, Y 8.264, Z 121.550}
   LaserEnd_Ext()
   LIN {X 11.720, Y 3.312, Z 121.550}
   LaserStart_Ext()
   LIN {X 11.720, Y -21.227, Z 121.550}
   LaserEnd_Ext()
   LIN {X 12.720, Y -19.877, Z 121.550}
   LaserStart_Ext()
   LIN {X 12.720, Y -3.058, Z 121.550}
   LaserEnd_Ext()
   LIN {X 10.153, Y -14.205, Z 122.400}
   LaserStart_Ext()
   LIN {X 10.446, Y -15.111, Z 122.400} C_DIS
   LIN {X 10.591, Y -16.451, Z 122.400} C_DIS
   LIN {X 10.389, Y -17.738, Z 122.400} C_DIS
   LIN {X 9.921, Y -18.802, Z 122.400} C_DIS
   LIN {X 8.966, Y -20.015, Z 122.400} C_DIS
   LIN {X 8.232, Y -20.558, Z 122.400} C_DIS
   LIN {X 5.789, Y -21.193, Z 122.400} C_DIS
   LIN {X 4.841, Y -21.302, Z 122.400} C_DIS
   LIN {X 4.004, Y -20.940, Z 122.400} C_DIS
   LIN {X 2.682, Y -20.413, Z 122.400} C_DIS
   LIN {X 1.904, Y -19.666, Z 122.400} C_DIS
   LIN {X 1.413, Y -19.004, Z 122.400} C_DIS
   LIN {X 0.766, Y -17.363, Z 122.400} C_DIS
   LIN {X 0.664, Y -16.399, Z 122.400} C_DIS
   LIN {X 0.919, Y -14.831, Z 122.400} C_DIS
   LIN {X 1.414, Y -13.749, Z 122.400} C_DIS
   LIN {X 2.274, Y -12.718, Z 122.400} C_DIS
   LIN {X 3.408, Y -11.911, Z 122.400} C_DIS
   LIN {X 4.025, Y -11.617, Z 122.400} C_DIS
   LIN {X 4.886, Y -11.554, Z 122.400} C_DIS
   LIN {X 6.408, Y -11.388, Z 122.400} C_DIS
   LIN {X 7.425, Y -11.808, Z 122.400} C_DIS
   LIN {X 8.683, Y -12.357, Z 122.400} C_DIS
   LIN {X 9.297, Y -13.038, Z 122.400} C_DIS
   LIN {X 10.153, Y -14.205, Z 122.400}
   LaserEnd_Ext()
   LIN {X 12.637, Y -21.769, Z 122.400}
   LaserStart_Ext()
   LIN {X 13.836, Y -19.997, Z 122.400} C_DIS
   LIN {X 14.194, Y -18.572, Z 122.400} C_DIS
   LIN {X 14.643, Y -16.275, Z 122.400} C_DIS
   LIN {X 14.627, Y -15.003, Z 122.400} C_DIS
   LIN {X 14.553, Y -11.939, Z 122.400} C_DIS
   LIN {X 14.492, Y -10.788, Z 122.400} C_DIS
   LIN {X 14.231, Y -6.857, Z 122.400} C_DIS
   LIN {X 14.205, Y -6.577, Z 122.400} C_DIS
   LIN {X 13.551, Y -1.161, Z 122.400} C_DIS
   LIN {X -0.961, Y 4.253, Z 122.400} C_DIS
   LIN {X -0.887, Y 0.589, Z 122.400} C_DIS
   LIN {X -0.906, Y 0.286, Z 122.400} C_DIS
   LIN {X -1.468, Y -5.765, Z 122.400} C_DIS
   LIN {X -1.579, Y -6.523, Z 122.400} C_DIS
   LIN {X -2.200, Y -10.163, Z 122.400} C_DIS
   LIN {X -2.501, Y -11.504, Z 122.400} C_DIS
   LIN {X -3.107, Y -14.151, Z 122.400} C_DIS
   LIN {X -3.172, Y -15.862, Z 122.400} C_DIS
   LIN {X -3.167, Y -18.356, Z 122.400} C_DIS
   LIN {X -2.442, Y -20.145, Z 122.400} C_DIS
   LIN {X -1.665, Y -21.688, Z 122.400} C_DIS
   LIN {X -0.063, Y -23.211, Z 122.400} C_DIS
   LIN {X 1.217, Y -24.238, Z 122.400} C_DIS
   LIN {X 3.120, Y -24.928, Z 122.400} C_DIS
   LIN {X 4.507, Y -25.300, Z 122.400} C_DIS
   LIN {X 6.510, Y -25.214, Z 122.400} C_DIS
   LIN {X 8.045, Y -25.013, Z 122.400} C_DIS
   LIN {X 9.895, Y -24.102, Z 122.400} C_DIS
   LIN {X 11.558, Y -23.088, Z 122.400} C_DIS
   LIN {X 12.637, Y -21.769, Z 122.400}
   LaserEnd_Ext()
   LIN {X 1.729, Y -23.360, Z 122.400}
   LaserStart_Ext()
   LIN {X 9.138, Y -23.360, Z 122.400}
   LaserEnd_Ext()
   LIN {X 10.831, Y -22.360, Z 122.400}
   LaserStart_Ext()
   LIN {X 0.493, Y -22.360, Z 122.400}
   LaserEnd_Ext()
   LIN {X -0.559, Y -21.360, Z 122.400}
   LaserStart_Ext()
   LIN {X 2.357, Y -21.360, Z 122.400}
   LaserEnd_Ext()
   LIN {X 8.829, Y -21.360, Z 122.400}
   LaserStart_Ext()
   LIN {X 11.679, Y -21.360, Z 122.400}
   LaserEnd_Ext()
   LIN {X 12.383, Y -20.360, Z 122.400}
   LaserStart_Ext()
   LIN {X 9.966, Y -20.360, Z 122.400}
   LaserEnd_Ext()
   LIN {X 1.185, Y -20.360, Z 122.400}
   LaserStart_Ext()
   LIN {X -1.214, Y -20.360, Z 122.400}
   LaserEnd_Ext()
   LIN {X -1.681, Y -19.360, Z 122.400}
   LaserStart_Ext()
   LIN {X 0.479, Y -19.360, Z 122.400}
   LaserEnd_Ext()
   LIN {X 10.750, Y -19.360, Z 122.400}
   LaserStart_Ext()
   LIN {X 12.965, Y -19.360, Z 122.400}
   LaserEnd_Ext()
   LIN {X 13.216, Y -18.360, Z 122.400}
   LaserStart_Ext()
   LIN {X 11.208, Y -18.360, Z 122.400}
   LaserEnd_Ext()
   LIN {X 0.084, Y -18.360, Z 122.400}
   LaserStart_Ext()
   LIN {X -2.086, Y -18.360, Z 122.400}
   LaserEnd_Ext()
   LIN {X -2.169, Y -17.360, Z 122.400}
   LaserStart_Ext()
   LIN {X -0.240, Y -17.360, Z 122.400}
   LaserEnd_Ext()
   LIN {X 11.460, Y -17.360, Z 122.400}
   LaserStart_Ext()
   LIN {X 13.412, Y -17.360, Z 122.400}
   LaserEnd_Ext()
   LIN {X 13.608, Y -16.360, Z 122.400}
   LaserStart_Ext()
   LIN {X 11.586, Y -16.360, Z 122.400}
   LaserEnd_Ext()
   LIN {X -0.334, Y -16.360, Z 122.400}
   LaserStart_Ext()
   LIN {X -2.171, Y -16.360, Z 122.400}
   LaserEnd_Ext()
   LIN {X -2.152, Y -15.360, Z 122.400}
   LaserStart_Ext()
   LIN {X -0.180, Y -15.360, Z 122.400}
   LaserEnd_Ext()
   LIN {X 11.479, Y -15.360, Z 122.400}
   LaserStart_Ext()
   LIN {X 13.631, Y -15.360, Z 122.400}
   LaserEnd_Ext()
   LIN {X 13.611, Y -14.360, Z 122.400}
   LaserStart_Ext()
   LIN {X 11.254, Y -14.360, Z 122.400}
   LaserEnd_Ext()
   LIN {X 0.035, Y -14.360, Z 122.400}
   LaserStart_Ext()
   LIN {X -2.115, Y -14.360, Z 122.400}
   LaserEnd_Ext()
   LIN {X -1.900, Y -13.360, Z 122.400}
   LaserStart_Ext()
   LIN {X 0.492, Y -13.360, Z 122.400}
   LaserEnd_Ext()
   LIN {X 10.774, Y -13.360, Z 122.400}
   LaserStart_Ext()
   LIN {X 13.587, Y -13.360, Z 122.400}
   LaserEnd_Ext()
   LIN {X 13.563, Y -12.360, Z 122.400}
   LaserStart_Ext()
   LIN {X 10.033, Y -12.360, Z 122.400}
   LaserEnd_Ext()
   LIN {X 1.270, Y -12.360, Z 122.400}
   LaserStart_Ext()
   LIN {X -1.671, Y -12.360, Z 122.400}
   LaserEnd_Ext()
   LIN {X -1.444, Y -11.360, Z 122.400}
   LaserStart_Ext()
   LIN {X 2.458, Y -11.360, Z 122.400}
   LaserEnd_Ext()
   LIN {X 8.899, Y -11.360, Z 122.400}
   LaserStart_Ext()
   LIN {X 13.521, Y -11.360, Z 122.400}
   LaserEnd_Ext()
   LIN {X 13.461, Y -10.360, Z 122.400}
   LaserStart_Ext()
   LIN {X -1.220, Y -10.360, Z 122.400}
   LaserEnd_Ext()
   LIN {X -1.048, Y -9.360, Z 122.400}
   LaserStart_Ext()
   LIN {X 13.395, Y -9.360, Z 122.400}
   LaserEnd_Ext()
   LIN {X 13.329, Y -8.360, Z 122.400}
   LaserStart_Ext()
   LIN {X -0.878, Y -8.360, Z 122.400}
   LaserEnd_Ext()
   LIN {X -0.707, Y -7.360, Z 122.400}
   LaserStart_Ext()
   LIN {X 13.262, Y -7.360, Z 122.400}
   LaserEnd_Ext()
   LIN {X 13.172, Y -6.360, Z 122.400}
   LaserStart_Ext()
   LIN {X -0.544, Y -6.360, Z 122.400}
   LaserEnd_Ext()
   LIN {X -0.426, Y -5.360, Z 122.400}
   LaserStart_Ext()
   LIN {X 13.051, Y -5.360, Z 122.400}
   LaserEnd_Ext()
   LIN {X 12.930, Y -4.360, Z 122.400}
   LaserStart_Ext()
   LIN {X -0.333, Y -4.360, Z 122.400}
   LaserEnd_Ext()
   LIN {X -0.240, Y -3.360, Z 122.400}
   LaserStart_Ext()
   LIN {X 12.809, Y -3.360, Z 122.400}
   LaserEnd_Ext()
   LIN {X 12.689, Y -2.360, Z 122.400}
   LaserStart_Ext()
   LIN {X -0.147, Y -2.360, Z 122.400}
   LaserEnd_Ext()
   LIN {X -0.054, Y -1.360, Z 122.400}
   LaserStart_Ext()
   LIN {X 11.223, Y -1.360, Z 122.400}
   LaserEnd_Ext()
   LIN {X 8.542, Y -0.360, Z 122.400}
   LaserStart_Ext()
   LIN {X 0.039, Y -0.360, Z 122.400}
   LaserEnd_Ext()
   LIN {X 0.112, Y 0.640, Z 122.400}
   LaserStart_Ext()
   LIN {X 5.862, Y 0.640, Z 122.400}
   LaserEnd_Ext()
   LIN {X 3.182, Y 1.640, Z 122.400}
   LaserStart_Ext()
   LIN {X 0.092, Y 1.640, Z 122.400}
   LaserEnd_Ext()
   LIN {X 0.072, Y 2.640, Z 122.400}
   LaserStart_Ext()
   LIN {X 0.501, Y 2.640, Z 122.400}
   LaserEnd_Ext()
   LIN {X 7.837, Y -20.758, Z 123.250}
   LaserStart_Ext()
   LIN {X 6.809, Y -21.025, Z 123.250} C_DIS
   LIN {X 4.923, Y -21.242, Z 123.250} C_DIS
   LIN {X 3.259, Y -20.522, Z 123.250} C_DIS
   LIN {X 2.666, Y -20.286, Z 123.250} C_DIS
   LIN {X 2.317, Y -19.951, Z 123.250} C_DIS
   LIN {X 1.227, Y -18.479, Z 123.250} C_DIS
   LIN {X 0.961, Y -17.806, Z 123.250} C_DIS
   LIN {X 0.749, Y -15.799, Z 123.250} C_DIS
   LIN {X 0.834, Y -15.276, Z 123.250} C_DIS
   LIN {X 1.760, Y -13.250, Z 123.250} C_DIS
   LIN {X 1.949, Y -13.024, Z 123.250} C_DIS
   LIN {X 3.919, Y -11.621, Z 123.250} C_DIS
   LIN {X 4.053, Y -11.589, Z 123.250} C_DIS
   LIN {X 6.471, Y -11.325, Z 123.250} C_DIS
   LIN {X 8.831, Y -12.354, Z 123.250} C_DIS
   LIN {X 10.364, Y -14.443, Z 123.250} C_DIS
   LIN {X 10.400, Y -14.553, Z 123.250} C_DIS
   LIN {X 10.651, Y -16.878, Z 123.250} C_DIS
   LIN {X 10.601, Y -17.197, Z 123.250} C_DIS
   LIN {X 9.729, Y -19.178, Z 123.250} C_DIS
   LIN {X 9.392, Y -19.606, Z 123.250} C_DIS
   LIN {X 7.837, Y -20.758, Z 123.250}
   LaserEnd_Ext()
   LIN {X 12.251, Y -22.324, Z 123.250}
   LaserStart_Ext()
   LIN {X 11.792, Y -22.886, Z 123.250} C_DIS
   LIN {X 9.246, Y -24.437, Z 123.250} C_DIS
   LIN {X 8.322, Y -24.893, Z 123.250} C_DIS
   LIN {X 5.855, Y -25.216, Z 123.250} C_DIS
   LIN {X 4.789, Y -25.262, Z 123.250} C_DIS
   LIN {X 2.497, Y -24.648, Z 123.250} C_DIS
   LIN {X 1.473, Y -24.276, Z 123.250} C_DIS
   LIN {X -0.644, Y -22.578, Z 123.250} C_DIS
   LIN {X -1.470, Y -21.793, Z 123.250} C_DIS
   LIN {X -2.716, Y -19.320, Z 123.250} C_DIS
   LIN {X -3.049, Y -18.495, Z 123.250} C_DIS
   LIN {X -3.057, Y -14.678, Z 123.250} C_DIS
   LIN {X -3.036, Y -14.108, Z 123.250} C_DIS
   LIN {X -2.264, Y -10.736, Z 123.250} C_DIS
   LIN {X -2.213, Y -10.511, Z 123.250} C_DIS
   LIN {X -1.813, Y -8.163, Z 123.250} C_DIS
   LIN {X 14.674, Y -14.313, Z 123.250} C_DIS
   LIN {X 14.715, Y -16.034, Z 123.250} C_DIS
   LIN {X 14.717, Y -16.196, Z 123.250} C_DIS
   LIN {X 14.107, Y -19.309, Z 123.250} C_DIS
   LIN {X 13.999, Y -19.742, Z 123.250} C_DIS
   LIN {X 12.251, Y -22.324, Z 123.250}
   LaserEnd_Ext()
   LIN {X 13.602, Y -16.687, Z 123.250}
   LaserStart_Ext()
   LIN {X 13.602, Y -14.980, Z 123.250}
   LaserEnd_Ext()
   LIN {X 12.602, Y -14.607, Z 123.250}
   LaserStart_Ext()
   LIN {X 12.602, Y -20.022, Z 123.250}
   LaserEnd_Ext()
   LIN {X 11.602, Y -21.499, Z 123.250}
   LaserStart_Ext()
   LIN {X 11.602, Y -17.268, Z 123.250}
   LaserEnd_Ext()
   LIN {X 11.602, Y -16.371, Z 123.250}
   LaserStart_Ext()
   LIN {X 11.602, Y -14.234, Z 123.250}
   LaserEnd_Ext()
   LIN {X 10.602, Y -19.665, Z 123.250}
   LaserStart_Ext()
   LIN {X 10.602, Y -22.440, Z 123.250}
   LaserEnd_Ext()
   LIN {X 9.602, Y -23.050, Z 123.250}
   LaserStart_Ext()
   LIN {X 9.602, Y -20.695, Z 123.250}
   LaserEnd_Ext()
   LIN {X 8.602, Y -21.435, Z 123.250}
   LaserStart_Ext()
   LIN {X 8.602, Y -23.640, Z 123.250}
   LaserEnd_Ext()
   LIN {X 7.602, Y -23.979, Z 123.250}
   LaserStart_Ext()
   LIN {X 7.602, Y -21.852, Z 123.250}
   LaserEnd_Ext()
   LIN {X 6.602, Y -22.055, Z 123.250}
   LaserStart_Ext()
   LIN {X 6.602, Y -24.110, Z 123.250}
   LaserEnd_Ext()
   LIN {X 5.602, Y -24.226, Z 123.250}
   LaserStart_Ext()
   LIN {X 5.602, Y -22.170, Z 123.250}
   LaserEnd_Ext()
   LIN {X 4.602, Y -22.188, Z 123.250}
   LaserStart_Ext()
   LIN {X 4.602, Y -24.176, Z 123.250}
   LaserEnd_Ext()
   LIN {X 3.602, Y -23.908, Z 123.250}
   LaserStart_Ext()
   LIN {X 3.602, Y -21.760, Z 123.250}
   LaserEnd_Ext()
   LIN {X 2.602, Y -10.877, Z 123.250}
   LaserStart_Ext()
   LIN {X 2.602, Y -11.331, Z 123.250}
   LaserEnd_Ext()
   LIN {X 2.602, Y -21.337, Z 123.250}
   LaserStart_Ext()
   LIN {X 2.602, Y -23.622, Z 123.250}
   LaserEnd_Ext()
   LIN {X 1.602, Y -23.097, Z 123.250}
   LaserStart_Ext()
   LIN {X 1.602, Y -20.649, Z 123.250}
   LaserEnd_Ext()
   LIN {X 1.602, Y -12.043, Z 123.250}
   LaserStart_Ext()
   LIN {X 1.602, Y -10.504, Z 123.250}
   LaserEnd_Ext()
   LIN {X 0.602, Y -10.131, Z 123.250}
   LaserStart_Ext()
   LIN {X 0.602, Y -13.378, Z 123.250}
   LaserEnd_Ext()
   LIN {X 0.602, Y -19.316, Z 123.250}
   LaserStart_Ext()
   LIN {X 0.602, Y -22.295, Z 123.250}
   LaserEnd_Ext()
   LIN {X -0.398, Y -21.432, Z 123.250}
   LaserStart_Ext()
   LIN {X -0.398, Y -9.758, Z 123.250}
   LaserEnd_Ext()
   LIN {X -1.398, Y -11.436, Z 123.250}
   LaserStart_Ext()
   LIN {X -1.398, Y -19.712, Z 123.250}
   LaserEnd_Ext()
   LIN {X 5.922, Y -23.782, Z 124.100}
   LaserStart_Ext()
   LIN {X 8.583, Y -24.774, Z 124.100} C_DIS
   LIN {X 5.200, Y -25.218, Z 124.100} C_DIS
   LIN {X 5.072, Y -25.223, Z 124.100} C_DIS
   LIN {X 1.874, Y -24.367, Z 124.100} C_DIS
   LIN {X 1.730, Y -24.315, Z 124.100} C_DIS
   LIN {X -1.225, Y -21.944, Z 124.100} C_DIS
   LIN {X -1.770, Y -20.914, Z 124.100} C_DIS
   LIN {X 5.922, Y -23.782, Z 124.100} C_DIS

   LaserOff_Ext()
   HALT

END
